	ELSIF byASCII=16#61 THEN	sOut_Single:='a';
	ELSIF byASCII=16#62 THEN  	sOut_Single:='b';
	ELSIF byASCII=16#63 THEN  	sOut_Single:='c';
	ELSIF byASCII=16#64 THEN	sOut_Single:='d';
	ELSIF byASCII=16#65 THEN	sOut_Single:='e';
	ELSIF byASCII=16#66 THEN	sOut_Single:='f';
	ELSIF byASCII=16#67 THEN	sOut_Single:='g';
	ELSIF byASCII=16#68 THEN	sOut_Single:='h';
	ELSIF byASCII=16#69 THEN	sOut_Single:='i';
	ELSIF byASCII=16#6A THEN	sOut_Single:='j';
	ELSIF byASCII=16#6B THEN	sOut_Single:='k';
	ELSIF byASCII=16#6C THEN	sOut_Single:='l';
	ELSIF byASCII=16#6D THEN	sOut_Single:='m';
	ELSIF byASCII=16#6E THEN	sOut_Single:='n';
	ELSIF byASCII=16#6F THEN	sOut_Single:='o';
	ELSIF byASCII=16#70 THEN	sOut_Single:='p';
	ELSIF byASCII=16#71 THEN	sOut_Single:='q';
	ELSIF byASCII=16#72 THEN	sOut_Single:='r';
	ELSIF byASCII=16#73 THEN	sOut_Single:='s';
	ELSIF byASCII=16#74 THEN	sOut_Single:='t';
	ELSIF byASCII=16#75 THEN	sOut_Single:='u';
	ELSIF byASCII=16#76 THEN	sOut_Single:='v';
	ELSIF byASCII=16#77 THEN	sOut_Single:='w';
	ELSIF byASCII=16#78 THEN	sOut_Single:='x';
	ELSIF byASCII=16#79 THEN	sOut_Single:='y';
	ELSIF byASCII=16#7A THEN	sOut_Single:='z';
	ELSIF byASCII=16#7B THEN	sOut_Single:='{';
	ELSIF byASCII=16#7C THEN	sOut_Single:='|';
	ELSIF byASCII=16#7D THEN	sOut_Single:='}';
	                                         
	ELSIF byASCII=16#30 THEN  	sOut_Single:='0';
	ELSIF byASCII=16#31 THEN  	sOut_Single:='1';
	ELSIF byASCII=16#32 THEN	sOut_Single:='2';
	ELSIF byASCII=16#33 THEN	sOut_Single:='3';
	ELSIF byASCII=16#34 THEN	sOut_Single:='4';
	ELSIF byASCII=16#35 THEN	sOut_Single:='5';
	ELSIF byASCII=16#36 THEN	sOut_Single:='6';
	ELSIF byASCII=16#37 THEN	sOut_Single:='7';
	ELSIF byASCII=16#38 THEN	sOut_Single:='8';
	ELSIF byASCII=16#39 THEN	sOut_Single:='9';
	ELSIF byASCII=16#3A THEN	sOut_Single:=':';
	ELSIF byASCII=16#3B THEN	sOut_Single:=';';
	ELSIF byASCII=16#3C THEN	sOut_Single:='<';
	ELSIF byASCII=16#3D THEN	sOut_Single:='=';
	ELSIF byASCII=16#3E THEN	sOut_Single:='>';
	ELSIF byASCII=16#3F THEN	sOut_Single:='?';
	ELSIF byASCII=16#40 THEN	sOut_Single:='@';
		                                     
	ELSIF byASCII=16#21 THEN	sOut_Single:='!';
	ELSIF byASCII=16#22 THEN	sOut_Single:='"';
	ELSIF byASCII=16#23 THEN	sOut_Single:='#';
//	ELSIF byASCII=16#24 THEN	sOut_Single:='$';
	ELSIF byASCII=16#25 THEN	sOut_Single:='%';
	ELSIF byASCII=16#26 THEN	sOut_Single:='&';
//	ELSIF byASCII=16#27 THEN	sOut_Single:=''';
	ELSIF byASCII=16#28 THEN	sOut_Single:='(';
	ELSIF byASCII=16#29 THEN	sOut_Single:=')';
	ELSIF byASCII=16#2A THEN	sOut_Single:='*';
	ELSIF byASCII=16#2B THEN	sOut_Single:='+';
	ELSIF byASCII=16#2C THEN	sOut_Single:=',';
	ELSIF byASCII=16#2D THEN	sOut_Single:='-';
	ELSIF byASCII=16#2E THEN	sOut_Single:='.';
	ELSIF byASCII=16#2F THEN	sOut_Single:='/';
	ELSE
		;	 //错误标志
	END_IF

END_FUNCTION_BLOCK

// Device/Application/PLC_PRG
PROGRAM PLC_PRG
VAR
	//(bHomingDone AND XRAY_RS485.Main_Step=20) OR Entity_IO.bEmergencyStop
	count: BYTE;
	bOver: BOOL; //关机结束指令
	bDebug_Laser:BOOL;
	TOF_Laser	:TOF;//激光灯控制
	TP_Laser	:TP;
	F_TRIG1		:F_TRIG;//激光灯按钮关闭
	R_TRIG1		:R_TRIG;//激光灯按钮关闭
	TOF_ET:TIME;
	TOF_PowerDelay: TOF;//延迟断电继电器控制
	LS_GetIPAddress_1: LS_GetIPAddress;
	LS_SetIPAddress_1: LS_SetIPAddress;
	rPLC_Load:REAL;
	LS_SetDintDT_1:LS_SysLib.LS_SetDintDT;
	bSetSysTime:BOOL;
	LS_ReadDintDT_1:LS_SysLib.LS_ReadDintDT;
	
	TON_StopScan:TON;

	iValidTrigger:UINT;
	iHopeNumPulse:UINT:=108;
	
	Step_Idle:INT;//待机模式下工作步骤
	Step_Scout:INT;//定位片模式下工作步骤
	Step_CBCT:INT;//CBCT模式下工作步骤
	Step_QuickScan:INT;//快速扫描下的工作步骤
	Step_DR:INT;//DR的工作步骤
	Step_XZ:INT;//XZ的工作步骤
	Step_AutoDR:INT;//自动空气校正DR
	bPulseOneStop	:BOOL;
	bScoutLast,bCBCTLast:BOOL;//最后一次扫描标志位

	TON_S30,TON_S40,TON_S41,TON_S42,TON_S43,TON_S50,TON_S52,TON_S60,TON_S70,TON_S80,TON_S90,TON_S44:TON;
	TON_S20_ABS,TON_S70_ABSX,TON_S70_ABSQ:TON;
	TOF_S40,TOF_S50:Standard.TOF;
	bXaryTwo_TEMP:BOOL; //二档输出中间变量
	
	TON_I00,TON_I10,TON_I20,TON_I30,TON_I40,TON_I50:Standard.TON;
	TON_C10,TON_C20,TON_C30,TON_C40,TON_C50,TON_C60,TON_C70,TON_C72,TON_C79,TON_C80,TON_C90,TON_C100,TON_C80_ABS,TON_C20_ABS:TON;
	TON_C210,TON_C201,TON_C220,TON_C230,TON_C240,TON_C250:TON;
	TOF_C80:Standard.TOF;
	R_TRIG_C20,R_TRIG_C220,R_TRIG_Jog,R_MoveRecordPos,R_RelStop:Standard.R_TRIG;
	F_TRIG_C20,F_TRIG_Jog:Standard.F_TRIG;
	
	AAA:STRING:='QWE';
	bSelfOK: BOOL;
	HandSelfStep: INT;
	bErrorReset:BOOL;
	TON_Error:TON;
	bHomingDone: BOOL;
	
	bGetPLC_IP,bSetPLC_IP,bGetPLC_Load:BOOL;
	
	TON_Home,TON_Home1:TON;
	
	bTestXayOne: BOOL;
	bTestXayTwo: BOOL;

	C_100: BOOL;
	bTCP_Socket:BOOL;
	TOF_JOG:TOF;
	bTestTrigger: BOOL;
	
	XZ_Velocity:REAL:=10;//设置不扫描时快速到扫描位的速度
	bTestTrigger11: BOOL;
	bTestTrigger22: BOOL;
	
	CTBOX_TON1:Standard.TON;
	CTBOX_TOF1:Standard.TOF;
	
	TON_IDLE:TON;
	bCBCT_AUTO_Manual:BOOL;//自动扫，手动扫标志位
	
	
	EncoderNum1,iStartTrigger1:UDINT;
	DB_EncoderNum1:UDINT;		//差值
	R_TRIG_debug,R_TRIG_debug2:R_TRIG;
	iActNumPulse1:UINT;//有效触发次数
	
	iSamplingRate1: INT:=2400;
	
	iHopePulse1:UINT;
	deubg_out:BOOL;
END_VAR

VAR PERSISTENT RETAIN
	rBedRecordHeight:REAL;//断电保存
	rBedRecordLength:REAL;//断电保存
END_VAR

VAR_OUTPUT	
	LampCmd5,LampCmd6,LampCmd7,LampCmd8:E_LampCmd;
END_VAR

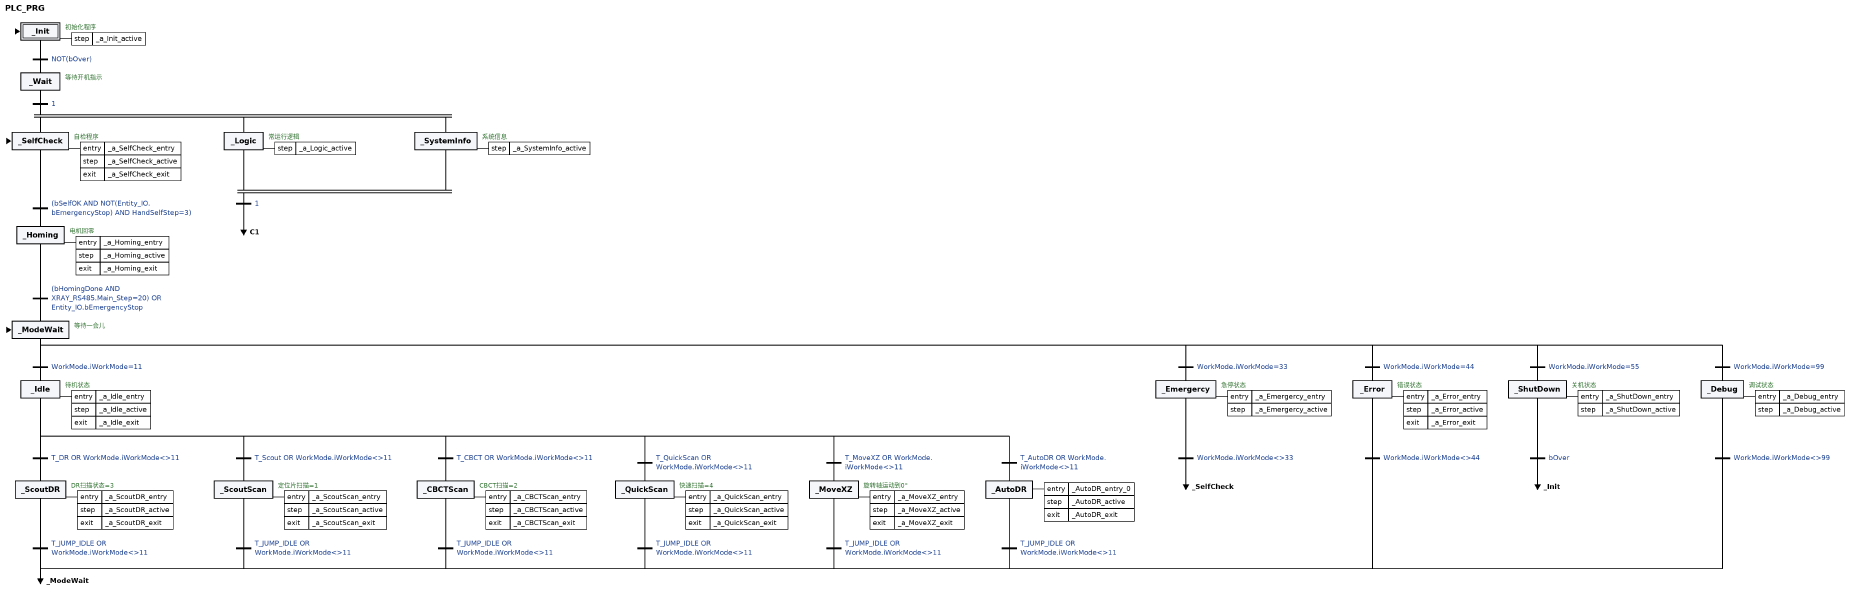
// 初始化程序
INITIAL_STEP _Init:
    _a_Init_active(N);  // step action
END_STEP
TRANSITION FROM _Init TO _Wait
    := NOT(bOver);
END_TRANSITION
// 等待开机指示
STEP _Wait:
END_STEP
TRANSITION FROM _Wait TO (_SelfCheck, _Logic, _SystemInfo)
    := 1;
END_TRANSITION
// 自检程序
STEP _SelfCheck:
    _a_SelfCheck_entry(P1);  // entry action
    _a_SelfCheck_active(N);  // step action
    _a_SelfCheck_exit(P0);  // exit action
END_STEP
TRANSITION FROM _SelfCheck TO _Homing
    := (bSelfOK AND NOT(Entity_IO.bEmergencyStop) AND HandSelfStep=3);
END_TRANSITION
// 电机回零
STEP _Homing:
    _a_Homing_entry(P1);  // entry action
    _a_Homing_active(N);  // step action
    _a_Homing_exit(P0);  // exit action
END_STEP
TRANSITION FROM _Homing TO _ModeWait
    := (bHomingDone AND XRAY_RS485.Main_Step=20) OR Entity_IO.bEmergencyStop;
END_TRANSITION
// 等待一会儿
STEP _ModeWait:
END_STEP
TRANSITION FROM _ModeWait TO _Idle
    := WorkMode.iWorkMode=11;
END_TRANSITION
// 待机状态
STEP _Idle:
    _a_Idle_entry(P1);  // entry action
    _a_Idle_active(N);  // step action
    _a_Idle_exit(P0);  // exit action
END_STEP
TRANSITION FROM _Idle TO _ScoutDR
    := T_DR OR WorkMode.iWorkMode<>11;
END_TRANSITION
// DR扫描状态=3
STEP _ScoutDR:
    _a_ScoutDR_entry(P1);  // entry action
    _a_ScoutDR_active(N);  // step action
    _a_ScoutDR_exit(P0);  // exit action
END_STEP
TRANSITION FROM _ScoutDR TO _ModeWait
    := T_JUMP_IDLE OR WorkMode.iWorkMode<>11;
END_TRANSITION
TRANSITION FROM _Idle TO _ScoutScan
    := T_Scout OR WorkMode.iWorkMode<>11;
END_TRANSITION
// 定位片扫描=1
STEP _ScoutScan:
    _a_ScoutScan_entry(P1);  // entry action
    _a_ScoutScan_active(N);  // step action
    _a_ScoutScan_exit(P0);  // exit action
END_STEP
TRANSITION FROM _ScoutScan TO _ModeWait
    := T_JUMP_IDLE OR WorkMode.iWorkMode<>11;
END_TRANSITION
TRANSITION FROM _Idle TO _CBCTScan
    := T_CBCT OR WorkMode.iWorkMode<>11;
END_TRANSITION
// CBCT扫描=2
STEP _CBCTScan:
    _a_CBCTScan_entry(P1);  // entry action
    _a_CBCTScan_active(N);  // step action
    _a_CBCTScan_exit(P0);  // exit action
END_STEP
TRANSITION FROM _CBCTScan TO _ModeWait
    := T_JUMP_IDLE OR WorkMode.iWorkMode<>11;
END_TRANSITION
TRANSITION FROM _Idle TO _QuickScan
    := T_QuickScan OR WorkMode.iWorkMode<>11;
END_TRANSITION
// 快速扫描=4
STEP _QuickScan:
    _a_QuickScan_entry(P1);  // entry action
    _a_QuickScan_active(N);  // step action
    _a_QuickScan_exit(P0);  // exit action
END_STEP
TRANSITION FROM _QuickScan TO _ModeWait
    := T_JUMP_IDLE OR WorkMode.iWorkMode<>11;
END_TRANSITION
TRANSITION FROM _Idle TO _MoveXZ
    := T_MoveXZ OR WorkMode.iWorkMode<>11;
END_TRANSITION
// 旋转轴运动到0°
STEP _MoveXZ:
    _a_MoveXZ_entry(P1);  // entry action
    _a_MoveXZ_active(N);  // step action
    _a_MoveXZ_exit(P0);  // exit action
END_STEP
TRANSITION FROM _MoveXZ TO _ModeWait
    := T_JUMP_IDLE OR WorkMode.iWorkMode<>11;
END_TRANSITION
TRANSITION FROM _Idle TO _AutoDR
    := T_AutoDR OR WorkMode.iWorkMode<>11;
END_TRANSITION
STEP _AutoDR:
    _AutoDR_entry_0(P1);  // entry action
    _AutoDR_active(N);  // step action
    _AutoDR_exit(P0);  // exit action
END_STEP
TRANSITION FROM _AutoDR TO _ModeWait
    := T_JUMP_IDLE OR WorkMode.iWorkMode<>11;
END_TRANSITION
TRANSITION FROM _ModeWait TO _Emergercy
    := WorkMode.iWorkMode=33;
END_TRANSITION
// 急停状态
STEP _Emergercy:
    _a_Emergercy_entry(P1);  // entry action
    _a_Emergercy_active(N);  // step action
END_STEP
TRANSITION FROM _Emergercy TO _SelfCheck
    := WorkMode.iWorkMode<>33;
END_TRANSITION
TRANSITION FROM _ModeWait TO _Error
    := WorkMode.iWorkMode=44;
END_TRANSITION
// 错误状态
STEP _Error:
    _a_Error_entry(P1);  // entry action
    _a_Error_active(N);  // step action
    _a_Error_exit(P0);  // exit action
END_STEP
TRANSITION FROM _Error TO _ModeWait
    := WorkMode.iWorkMode<>44;
END_TRANSITION
TRANSITION FROM _ModeWait TO _ShutDown
    := WorkMode.iWorkMode=55;
END_TRANSITION
// 关机状态
STEP _ShutDown:
    _a_ShutDown_entry(P1);  // entry action
    _a_ShutDown_active(N);  // step action
END_STEP
TRANSITION FROM _ShutDown TO _Init
    := bOver;
END_TRANSITION
TRANSITION FROM _ModeWait TO _Debug
    := WorkMode.iWorkMode=99;
END_TRANSITION
// 调试状态
STEP _Debug:
    _a_Debug_entry(P1);  // entry action
    _a_Debug_active(N);  // step action
END_STEP
TRANSITION FROM _Debug TO _ModeWait
    := WorkMode.iWorkMode<>99;
END_TRANSITION
// 常运行逻辑
STEP _Logic:
    _a_Logic_active(N);  // step action
END_STEP
// 系统信息
STEP _SystemInfo:
    _a_SystemInfo_active(N);  // step action
END_STEP
TRANSITION FROM (_Logic, _SystemInfo) TO (_Logic, _SystemInfo)
    := 1;
END_TRANSITION
// branch label C1
// branch label B1

ACTION _a_SelfCheck_active:

GVL_State.iPLC_State:=20;

(*目前只检查电机错误*)
	bSelfOK:=NOT(Axis_QJ.QJ_AxisState.bAxisErr OR Axis_XZ.XZ_AxisState.bAxisErr);

(*有错误自动复位*)	
	IF Entity_IO.bEmergencyStop = FALSE  THEN  //急停未被拍下
		CASE HandSelfStep OF
			0:
				IF Axis_QJ.QJ_AxisState.bAxisErr THEN
					Axis_QJ.QJ_AxisCmd.bReset:=TRUE;
				ELSE
					HandSelfStep:=1;
				END_IF
				
			1:
				IF Axis_XZ.XZ_AxisState.bAxisErr THEN
					Axis_XZ.XZ_AxisCmd.bReset:=TRUE;
				ELSE
					HandSelfStep:=2;
				END_IF
				
			2:
				Axis_XZ.XZ_AxisCmd.bReset:=FALSE;
				Axis_QJ.QJ_AxisCmd.bReset:=FALSE;
				HandSelfStep:=3;
				
			3:
				;	
		END_CASE
	END_IF;
	
(*旋转电机写入电机回零默认参数*)
	Axis_XZ.XZ_AxisCmd.AxisPara.rHomeAcc:=5.0;
	Axis_XZ.XZ_AxisCmd.AxisPara.iHomeMode:=10;
	Axis_XZ.XZ_AxisCmd.AxisPara.rHomeHighSpeed:=10;
	Axis_XZ.XZ_AxisCmd.AxisPara.rHomeLowSpeed:=5;
	
(*前进写入电机回零默认参数*)
	Axis_QJ.QJ_AxisCmd.AxisPara.rHomeAcc:=5.0;
	Axis_QJ.QJ_AxisCmd.AxisPara.iHomeMode:=10;
	Axis_QJ.QJ_AxisCmd.AxisPara.rHomeHighSpeed:=10;
	Axis_QJ.QJ_AxisCmd.AxisPara.rHomeLowSpeed:=5;
END_ACTION

ACTION _a_MoveXZ_entry:

GVL_State.iPLC_State:=52;//告诉上位机52，机架运动到位0位置
Step_XZ:=0; 
bTCP_Socket:=TRUE;
GVL_SCAN.bEnableScout:=FALSE;
GVL_SCAN.bEnableTrigger:=FALSE;
END_ACTION

ACTION _a_QuickScan_exit:


	LampCmd5:=E_LampCmd.关闭;
	LampCmd6:=E_LampCmd.关闭;
	LampCmd7:=E_LampCmd.关闭;
	LampCmd8:=E_LampCmd.关闭;
	
	Entity_IO.bTriggerPannel:=FALSE;
	Entity_IO.bTriggerOut:=FALSE;
	
	GVL_State.bEnable_CTBOX:=FALSE;//关闭CTBOX发送灯使能
END_ACTION

TRANSITION T_JUMP_IDLE:


	(*跳转到待机指令*)
	(*1.手动终止扫描，上位机发送终止扫描，扫描结束*)
	TON_StopScan.Q 
	OR (WorkStation_TCP.PLC_RECV1.m_nControlState>=1 AND WorkStation_TCP.PLC_RECV1.m_nSocketType=1)
	OR GVL_SCAN.bJumpScan;
END_TRANSITION

ACTION _a_ScoutDR_active:


	CASE Step_DR OF
		0:	//初始化准备流程
			(*1.给上位机发送的数据*)
			WorkStation_TCP.PLC_SEND1.m_nMoveState:=0;			//send[9]
			Axis_XZ.XZ_AxisCmd.bAbs:=FALSE;
			bTCP_Socket:=FALSE;
			bScoutLast := FALSE;
			
			(*2.运动准备数据*)
			(*2.1 写入旋转速度参数*)
			Axis_XZ.XZ_AxisCmd.AxisPara.rAbsVelocity:=36;//定位像扫描按照设定速度运动
			
			TON_S20_ABS(IN:=FALSE);
			Step_DR:=10;
		
		10:	//运动过程中变量复位标志
			TON_S30(IN:= FALSE );
			TON_S40(IN:= FALSE);TON_S50(IN:= FALSE);
			TON_S70(IN:= FALSE);TON_S80(IN:= FALSE);
			TOF_S50(IN:= FALSE);TON_S60(IN:= FALSE);
			TON_S52(IN:= FALSE );TON_S41(IN:=FALSE);
			TON_S43(IN:= FALSE );TON_S20_ABS(IN:=FALSE);	
			Axis_XZ.XZ_AxisCmd.bAbs:=FALSE;
			Step_DR:=20;
			
		20://开启运动
			(*1.给上位机发送的数据*)
			WorkStation_TCP.PLC_SEND1.m_nExpStates	:=1;//为曝光状态，枚举值，0:idle（空闲） 1:prep（训机） 2: ready（训机结束，准备完成，可以出束） 3: XrayOn（出射线） 4:XrayOff（关射线） 5 error；
			WorkStation_TCP.PLC_SEND1.m_nMoveState	:=0;//起始、终止状态， 默认值-1， 0为当前扫描方案（与常规意义不同，注意区别）处于准备好状态，可以准备扫描；1为当前扫描方案结束，运动过程中值为-1
			WorkStation_TCP.PLC_SEND1.m_nScanProType:=2;//执行扫描方案的类型，0为自动扫描，1为手动扫描，2为无设置意义的值，默认值为2
	
			(*2.旋转轴运动*)
			Axis_XZ.XZ_AxisCmd.AxisPara.rAbsPosition:=LIMIT(-4,WorkStation_TCP.PLC_RECV1.m_nRotateBegin,363);
			TON_S20_ABS(IN:= TRUE, PT:=T#1S );
			Axis_XZ.XZ_AxisCmd.bAbs:=TON_S20_ABS.Q;
			
			(*3.跳转下一个步骤*)	
			IF  ABS(Axis_XZ.XZ_AxisState.rActPosition-WorkStation_TCP.PLC_RECV1.m_nRotateBegin)<=1 THEN 
				Step_DR:=21;
			END_IF
				
		21://射线源参数写入成功标志
			TON_S20_ABS(IN:=FALSE);
			Axis_XZ.XZ_AxisCmd.bAbs:=FALSE;
			IF XRAY_RS485.Standby_Step=60 THEN		(*增加射线源参数写入成功标志*)
				Step_DR:=30;
			END_IF

		30: //开启7灯闪烁
			(*1.给上位机数据*)
			WorkStation_TCP.PLC_SEND1.m_nMoveState:=1;			//send[9]
			TON_S30(IN:=TRUE , PT:=T#1S , Q=> , ET=> );
			
			(*2.7灯闪烁*)
			GVL_State.bEnable_CTBOX:=TRUE;//开启CTBOX发送灯的状态
			LampCmd7:=E_LampCmd.慢闪;
			WorkStation_TCP.PLC_SEND1.m_nFocus:=7;//按键提示0228
			
			(*3.跳转*)
			IF TON_S30.Q THEN
				Step_DR:=31;
			END_IF
			
		31:
			GVL_State.bEnable_CTBOX:=FALSE;//关闭CTBOX发送灯的状态
			Step_DR:=40;
		
		40://等待用户按7键。此时7灯一直在闪烁
			(*1.发送上位机状态*)
			IF CTBOX_RS232.CTBOX_KEY_Manual THEN
				WorkStation_TCP.PLC_SEND1.m_nScanProType:=1;//执行扫描方案的类型，0为自动扫描，1为手动扫描，2为无设置意义的值，默认值为2
			END_IF
			
			(*2.7灯关闭*)
			TON_S41(IN:=(WorkStation_TCP.PLC_SEND1.m_nScanProType=1) , PT:=T#100MS , Q=> , ET=> );
			IF TON_S41.Q THEN
				LampCmd7:=E_LampCmd.关闭;  		//7灯关闭
				WorkStation_TCP.PLC_SEND1.m_nFocus:=0;//关闭按键提示0228
			END_IF
			
			TON_S42(IN:=FALSE , Q=> , ET=> );	//复位
			TON_S43(IN:=FALSE , Q=> , ET=> );	//复位
			
			(*3.跳转*)
			TON_S40(IN:= (WorkStation_TCP.PLC_SEND1.m_nScanProType=1), PT:=T#1S , Q=> , ET=> );
			IF TON_S40.Q THEN
				Step_DR:=41;
			END_IF
			
		41://中间状态清零，特别是从80跳转过来的变量清零
			GVL_State.bEnable_CTBOX:=FALSE;//关闭CTBOX发送灯的状态
			TON_S41(IN:=FALSE);TON_S80(IN:=FALSE);
			Entity_IO.bXaryOne:=FALSE;
			GVL_SCAN.bEnableTrigger:=FALSE;
			GVL_State.bScoutSecond:=TRUE;
			IF XRAY_RS485.Standby_Step=60 THEN
				Step_DR:=42;
			END_IF;	

		42:
			(*1.开启透视*)
			Entity_IO.bXaryOne:=TRUE;		//开启透视
			
			IF ABS(Axis_XZ.XZ_AxisState.rActPosition-WorkStation_TCP.PLC_RECV1.m_nAngleStart)<1 THEN
				GVL_SCAN.bEnableScout:=TRUE;	
			ELSE
				GVL_SCAN.bEnableScout:=FALSE;
			END_IF
			
			(*2.跳转指令*)
			TON_S43(IN:= Entity_IO.bXaryOne, PT:=T#1S , Q=> , ET=> );
			IF TON_S43.Q THEN
				IF XRAY_RS485.Rad_Step>=20 THEN  //此时射线源收到  =20
					Step_DR:=50;
				END_IF
			ELSE
			;
			END_IF;
			
			(*3.判断是否最后一次扫描标志位*)
			IF WorkStation_TCP.PLC_RECV1.m_nLastMsg=1 THEN
				bScoutLast := TRUE;
			ELSE
				bScoutLast := FALSE;
			END_IF 
			
			(*4.一二档信号超时报警，射线源30秒连续开启曝光会报警*)
			TON_S42(IN:=Entity_IO.bXaryOne , PT:=T#60S , Q=> , ET=> );
			IF TON_S42.Q THEN
				Step_DR:=44;	
			END_IF
			
		44:
			Entity_IO.bXaryOne:=FALSE;
			GVL_SCAN.bJumpScan:=TRUE;		//结束扫描，射线源超时报警了，EL019，结束扫描
			Step_DR:=44;	

		50://固定位置直接曝光28次
			TON_S43(IN:=FALSE , Q=> , ET=> );	//复位
			(*1.发送给上位机的数据*)
			WorkStation_TCP.PLC_SEND1.m_nMoveState	:=2;			//send[9]//0-准备过程中 1-准备完成 2-曝光中 3-本次扫描结束	
			WorkStation_TCP.PLC_SEND1.m_nScanProType:=2;			//send[16]
			
			(*2.开启允许曝光指令*)
			IF Entity_IO.bXaryOne AND ABS(Axis_XZ.XZ_AxisState.rActPosition-WorkStation_TCP.PLC_RECV1.m_nAngleStart)<1 THEN //新增射线源状态位置
				GVL_SCAN.bEnableTrigger:=TRUE;
			ELSE
				GVL_SCAN.bEnableTrigger:=FALSE;
			END_IF
			
			(*3.此过程给固定时间4秒,处理扫描*)
			TON_S50(IN:=TRUE , PT:=T#4S);
			IF TON_S50.Q THEN
				Step_DR:=52;	
			END_IF
		
		52://出射线状态结束，采集射线源状态机信息 //增加2档信号8秒计时器清零操作
			TON_S52(IN:=NOT(Trigger_HaoboPannel.bScoutPulse) , PT:= T#3S );
			Entity_IO.bXaryOne:=NOT(TON_S52.Q);
			IF TON_S52.Q THEN
				IF XRAY_RS485.Main_Step=20 THEN
					Step_DR:=60;
				END_IF
			END_IF
			
		60://判断是否最后一次扫描，如是，直接跳到待机模式，如果不是，接着定位扫描 ，第一次定位像和第二次定位像不一样，增加了床的运动
			TON_S80(IN:=FALSE);
			Entity_IO.bXaryOne:=FALSE;
			Axis_QJ.QJ_AxisCmd.bAbs:=FALSE;
			Axis_XZ.XZ_AxisCmd.bAbs:=FALSE;	
			TON_S70_ABSQ(IN:=FALSE);TON_S70_ABSX(IN:=FALSE);
			TON_S60(IN:=TRUE , PT:=T#1600MS , Q=> , ET=> );//留些时间给上位机发送本次扫描结束方案标志
			WorkStation_TCP.PLC_SEND1.m_nMoveState:=3;		//send[9] //0-准备过程中 1-准备完成 2-曝光中 3-本次扫描结束	
			IF TON_S60.Q THEN
				IF (WorkStation_TCP.PLC_RECV1.m_nCircleIndex+1)>=(WorkStation_TCP.PLC_RECV1.m_nCircleCount) AND bScoutLast THEN 	//用于区分自动扫是否最后一次，此时=1，=1都等于1
					GVL_SCAN.bJumpScan:=TRUE;
				END_IF;
			END_IF
			
			IF WorkStation_TCP.PLC_RECV1.m_nSocketType=1 THEN //增加第二次运动判断，m_nSocketType=1 
				Step_DR:=70;
			END_IF
			
		70://上位机选择移动床位置，机架根据命令运动到位
			Axis_QJ.QJ_AxisCmd.AxisPara.rAbsPosition:=LIMIT(0,WorkStation_TCP.PLC_RECV1.m_fScanTop,900);
			Axis_QJ.QJ_AxisCmd.AxisPara.rAbsVelocity:=50; //单位mm/s
			TON_S70_ABSQ(IN:=TRUE , PT:=T#1S , Q=> , ET=> );
			Axis_QJ.QJ_AxisCmd.bAbs:=TON_S70_ABSQ.Q;
			
			Axis_XZ.XZ_AxisCmd.AxisPara.rAbsPosition:=LIMIT(-4,WorkStation_TCP.PLC_RECV1.m_nRotateBegin,363);
			TON_S70_ABSX(IN:=TRUE , PT:=T#1S , Q=> , ET=> );
			Axis_XZ.XZ_AxisCmd.bAbs:=TON_S70_ABSX.Q;
			
			IF ABS(Axis_QJ.QJ_AxisState.rActPosition-WorkStation_TCP.PLC_RECV1.m_fScanTop)<1 AND ABS(Axis_XZ.XZ_AxisState.rActPosition-WorkStation_TCP.PLC_RECV1.m_nRotateBegin)<1 THEN
				WorkStation_TCP.PLC_SEND1.m_nMoveState:=1;		//send[9] //0-准备过程中 1-准备完成 2-曝光中 3-本次扫描结束	
			ELSE
				WorkStation_TCP.PLC_SEND1.m_nMoveState:=0;		//send[9] //0-准备过程中 1-准备完成 2-曝光中 3-本次扫描结束	
			END_IF
			
			TON_S70(IN:=ABS(Axis_QJ.QJ_AxisState.rActPosition-WorkStation_TCP.PLC_RECV1.m_fScanTop)<1 
					AND ABS(Axis_XZ.XZ_AxisState.rActPosition-WorkStation_TCP.PLC_RECV1.m_nRotateBegin)<1, 
					PT:=T#2S , Q=> , ET=> );//给你2秒走到位
			IF TON_S70.Q THEN
				Step_DR:=80;
			END_IF
		
		80://准备跳转，中间变量复位
			TOF_S50(IN:= FALSE);TON_S60(IN:= FALSE);TON_S70(IN:= FALSE);
			TON_S41(IN:= FALSE);TON_S42(IN:= FALSE);
			TON_S70_ABSQ(IN:=FALSE);TON_S70_ABSX(IN:=FALSE);
			Axis_QJ.QJ_AxisCmd.bAbs:=FALSE;
			Axis_XZ.XZ_AxisCmd.bAbs:=FALSE;
			TON_S80(IN:=TRUE , PT:= T#1S, Q=> , ET=> );
			IF TON_S80.Q THEN
				Step_DR:=41;
			END_IF;	
	END_CASE
END_ACTION

ACTION _a_Idle_exit:


	Step_Idle:=0;
	
	LampCmd5:=E_LampCmd.关闭;
	LampCmd6:=E_LampCmd.关闭;
	LampCmd7:=E_LampCmd.关闭;
	LampCmd8:=E_LampCmd.关闭;
	
	GVL_State.bBooting:=FALSE;
END_ACTION

TRANSITION T_DR:

(*进入dr扫描*)
	WorkStation_TCP.PLC_RECV1.m_nSocketType=1 AND WorkStation_TCP.PLC_RECV1.m_nExpId=3
END_TRANSITION

ACTION _AutoDR_exit:


	LampCmd5:=E_LampCmd.关闭;
	LampCmd6:=E_LampCmd.关闭;
	LampCmd7:=E_LampCmd.关闭;
	LampCmd8:=E_LampCmd.关闭;
	
	Entity_IO.bTriggerPannel:=FALSE;
	Entity_IO.bTriggerOut:=FALSE;
END_ACTION

ACTION _a_Idle_entry:


	Step_Idle:=0; //
	bPulseOneStop:=TRUE;
	
	GVL_SCAN.bJumpScan:=FALSE;
	
	Axis_XZ.XZ_AxisCmd.bAbs:=FALSE;
	Axis_QJ.QJ_AxisCmd.bAbs:=FALSE;
	
	Axis_QJ.QJ_AxisCmd.bStop:=FALSE;
	Axis_XZ.XZ_AxisCmd.bStop:=FALSE;
		
	Axis_XZ.XZ_AxisCmd.bReset:=FALSE;
	Axis_QJ.QJ_AxisCmd.bReset:=FALSE;
	
	GVL_SCAN.bEnableTrigger:=FALSE;
	GVL_State.bBooting:=TRUE;
	
	WorkStation_TCP.PLC_SEND1.m_nFocus:=0;//按键提示

	Step_CBCT:=0;
	Step_Scout:=0;
END_ACTION

ACTION _a_SelfCheck_exit:


Axis_QJ.QJ_AxisCmd.bSetHomePara:=TRUE;

Axis_XZ.XZ_AxisCmd.bSetHomePara:=TRUE;
END_ACTION

ACTION _a_Error_entry:

	bErrorReset:=TRUE;
	TON_Error(IN:=FALSE);
END_ACTION

TRANSITION T_QuickScan:


(*进入快速扫描*)
	WorkStation_TCP.PLC_RECV1.m_nSocketType=1 AND WorkStation_TCP.PLC_RECV1.m_nExpId=4 //这里需要上位机增加一个4,判断是快速扫描
END_TRANSITION

ACTION _AutoDR_active:

	CASE Step_AutoDR OF 
		0:	//初始化准备流程
			(*1.给上位机发送的数据*)
			WorkStation_TCP.PLC_SEND1.m_nMoveState:=0;			//send[9] //0-准备过程中 1-准备完成 2-曝光中 3-本次扫描结束
			bTCP_Socket:=FALSE; 
			bCBCTLast:=FALSE;
			
			(*2.运动准备数据*)
			(*2.1 写入旋转速度参数*)
		(*	IF WorkStation_TCP.PLC_RECV1.m_fSecondPerCicle<>0 THEN//避免除零
				Axis_XZ.XZ_AxisCmd.AxisPara.rAbsVelocity:=UDINT_TO_REAL(LIMIT(360/300 ,360/WorkStation_TCP.PLC_RECV1.m_fSecondPerCicle ,360/20 ));
				XZ_Velocity:=LIMIT(360/300 ,360/UDINT_TO_REAL(WorkStation_TCP.PLC_RECV1.m_fSecondPerCicle) ,360/20);
			ELSE
				Axis_XZ.XZ_AxisCmd.AxisPara.rAbsVelocity:=8;
			END_IF;
		*)
			Axis_XZ.XZ_AxisCmd.AxisPara.rAbsVelocity:=36;
			Step_AutoDR:=10;

		10:	//运动过程中变量复位标志
			TON_C20(IN:= FALSE);TON_C30(IN:= FALSE);
			TON_C40(IN:= FALSE);TON_C50(IN:= FALSE);TON_C60(IN:= FALSE);
			TON_C70(IN:= FALSE);TON_C80(IN:= FALSE);TON_C72(IN:=FALSE);
			TON_C210(IN:= FALSE);TON_C220(IN:= FALSE);TON_C230(IN:= FALSE);
			TON_C240(IN:= FALSE);TON_C250(IN:= FALSE);
			TON_C20_ABS(IN:=FALSE);
			TOF_C80(IN:= FALSE);
			Axis_XZ.XZ_AxisCmd.bAbs:=FALSE;
			Step_AutoDR:=20;
			
		20://按5键，移动床到预设位置，松开即停，机架直接到预设位置
			(*1.发送给上位机的数据*)
			WorkStation_TCP.PLC_SEND1.m_nExpStates:=1;		//0-准备过程中 1-准备完成 2-曝光中 3-本次扫描结束	
			WorkStation_TCP.PLC_SEND1.m_nMoveState:=0;		//起始、终止状态， 默认值0， 1为当前扫描方案处于准备好状态，可以准备扫描；2为当前扫描方案结束，运动过程中值为0
			WorkStation_TCP.PLC_SEND1.m_nScanProType:=2;	//扫描方案类型 , 1-手动，0-自动. 
			
			(*2.旋转轴直接运动到目标位置*)
			Axis_XZ.XZ_AxisCmd.AxisPara.rAbsPosition:=LIMIT(-3,WorkStation_TCP.PLC_RECV1.m_nRotateBegin,363);
			Axis_XZ.XZ_AxisCmd.AxisPara.rAbsVelocity:=36;
			TON_C20_ABS(IN:=TRUE , PT:=T#1S);
			Axis_XZ.XZ_AxisCmd.bAbs:=TON_C20_ABS.Q;
			
			(*3.前进轴运动*)
			R_TRIG_C20(CLK:= CTBOX_RS232.CTBOX_KEY_MoveDistance, Q=> );//触发运动
			F_TRIG_C20(CLK:= CTBOX_RS232.CTBOX_KEY_MoveDistance, Q=> );//触发停止
			
			Axis_QJ.QJ_AxisCmd.bAbs	:=R_TRIG_C20.Q;
			Axis_QJ.QJ_AxisCmd.AxisPara.rAbsPosition	:=LIMIT(0,WorkStation_TCP.PLC_RECV1.m_fScanTop,900);
			Axis_QJ.QJ_AxisCmd.bStop:=F_TRIG_C20.Q;
			
			(*4.5灯逻辑处理*)
			GVL_State.bEnable_CTBOX:=TRUE;//开启CTBOX发送灯使能
			IF ABS(Axis_QJ.QJ_AxisState.rActPosition-WorkStation_TCP.PLC_RECV1.m_fScanTop)>1 THEN
				LampCmd5:=E_LampCmd.慢闪;
				WorkStation_TCP.PLC_SEND1.m_nFocus:=5;//按键提示0228
			ELSE
				LampCmd5:=E_LampCmd.关闭;
				WorkStation_TCP.PLC_SEND1.m_nFocus:=0;//关闭按键提示0228
			END_IF
			
			(*5.跳转*)
			TON_C20(IN:=ABS(Axis_QJ.QJ_AxisState.rActPosition-WorkStation_TCP.PLC_RECV1.m_fScanTop)<1 
				AND ABS(Axis_XZ.XZ_AxisState.rActPosition-WorkStation_TCP.PLC_RECV1.m_nRotateBegin)<1 , PT:=T#2S);
			IF TON_C20.Q THEN  
				Step_AutoDR:=30;
			END_IF
			
		30:	//射线源参数写入成功标志
			TON_C20_ABS(IN:=FALSE);
			LampCmd5:=E_LampCmd.关闭;
			Axis_XZ.XZ_AxisCmd.bAbs:=FALSE;
			Axis_QJ.QJ_AxisCmd.bAbs:=FALSE;
			Axis_QJ.QJ_AxisCmd.bStop:=FALSE;
			IF XRAY_RS485.Standby_Step=60 THEN
				Step_AutoDR:=40;
			END_IF
			
		40:	//7灯和8灯开始慢闪
			WorkStation_TCP.PLC_SEND1.m_nMoveState:=1;		//起始、终止状态， 默认值0， 1为当前扫描方案处于准备好状态
			LampCmd7:=E_LampCmd.慢闪;
			LampCmd8:=E_LampCmd.慢闪;
			WorkStation_TCP.PLC_SEND1.m_nFocus:=8;//按键提示0228
			TON_C40(IN:=TRUE , PT:=T#600MS , Q=> , ET=> );
			IF TON_C40.Q THEN
				Step_AutoDR:=41;
			END_IF
		41:
			GVL_State.bEnable_CTBOX:=FALSE;//开启CTBOX发送灯使能
			Step_AutoDR:=50;
			
		50://用户选择自动扫描或手动扫描
			IF CTBOX_RS232.CTBOX_KEY_Auto=FALSE AND CTBOX_RS232.CTBOX_KEY_Manual THEN
				WorkStation_TCP.PLC_SEND1.m_nScanProType:=1;								//扫描方案类型 , 1-手动，0-自动. 
				bCBCT_AUTO_Manual:=TRUE;
			ELSIF CTBOX_RS232.CTBOX_KEY_Auto AND CTBOX_RS232.CTBOX_KEY_Manual=FALSE THEN
				WorkStation_TCP.PLC_SEND1.m_nScanProType:=0;								//扫描方案类型 , 1-手动，0-自动. 
				bCBCT_AUTO_Manual:=FALSE;
			ELSIF CTBOX_RS232.CTBOX_KEY_Auto=FALSE AND CTBOX_RS232.CTBOX_KEY_Manual=FALSE THEN
				;
			ELSIF CTBOX_RS232.CTBOX_KEY_Auto AND CTBOX_RS232.CTBOX_KEY_Manual THEN
				;
			END_IF
			
			IF (CTBOX_RS232.CTBOX_KEY_Auto AND CTBOX_RS232.CTBOX_KEY_Manual=FALSE) OR CTBOX_RS232.CTBOX_KEY_Manual AND CTBOX_RS232.CTBOX_KEY_Auto=FALSE THEN
				Step_AutoDR:=60;
			END_IF
			
		60://7和8灯关闭 
			GVL_State.bEnable_CTBOX:=TRUE;
			LampCmd7:=E_LampCmd.关闭;
			LampCmd8:=E_LampCmd.关闭;
			WorkStation_TCP.PLC_SEND1.m_nFocus:=0;	//关闭按键提示0228
			TON_C60(IN:= TRUE, PT:=T#1S , Q=> , ET=> );
			
			IF TON_C60.Q THEN
				Step_AutoDR:=70;
			END_IF
			
		70://扫描中间态，给跳转用的
			GVL_State.bEnable_CTBOX:=FALSE;//关闭CTBOX发送灯使能
			WorkStation_TCP.PLC_SEND1.m_nMoveState	:=1;	//send[9]
			WorkStation_TCP.PLC_SEND1.m_nScanProType:=2;	//send[16]
			TON_C70(IN:=TRUE , PT:=T#2S , Q=> , ET=> );
			TON_C220(IN:=FALSE);TON_C72(IN:=FALSE);TON_S50(IN:=FALSE , PT:=T#4S);
			Axis_QJ.QJ_AxisCmd.bAbs:=FALSE;//复位前进轴
			Axis_XZ.XZ_AxisCmd.bAbs:=FALSE;//复位旋转轴
			TON_C72(IN:=FALSE);
			TON_C79(IN:=TRUE , PT:= T#1S, Q=> , ET=> );
			
			IF XRAY_RS485.Standby_Step=60 THEN  //保证写入参数
				Entity_IO.bXaryOne:=TRUE;//开启透视
			END_IF;
			
			(*判断是否最后一次扫描*)
			IF WorkStation_TCP.PLC_RECV1.m_nLastMsg=1 THEN
				bCBCTLast := TRUE;
			ELSE
				bCBCTLast := FALSE;
			END_IF
			
			(*跳转指令*)
			IF TON_C70.Q AND Entity_IO.bXaryOne THEN
				Step_AutoDR:=79;
			END_IF
			
		74:
			Entity_IO.bXaryOne:=FALSE;
			GVL_SCAN.bJumpScan:=TRUE;		//结束扫描，射线源超时报警了，EL019，结束扫描
			Step_AutoDR:=74;
			
		79:
			Axis_XZ.XZ_AxisCmd.bAbs:=FALSE;
			TON_C80_ABS(IN:=FALSE);
			TON_S50(IN:=FALSE , PT:=T#4S);
			TON_C79(IN:=TRUE , PT:= T#4S, Q=> , ET=> );
			IF TON_C79.Q THEN
				Step_AutoDR:=80;
			END_IF
			
			IF ABS(Axis_XZ.XZ_AxisState.rActPosition-WorkStation_TCP.PLC_RECV1.m_nAngleStart)<1 THEN
				GVL_SCAN.bEnableScout:=TRUE;	
			ELSE
				GVL_SCAN.bEnableScout:=FALSE;
			END_IF
			
		80://第一次自动扫描
			(*1.给上位机发送的数*)
			TON_C79(IN:=FALSE);
			WorkStation_TCP.PLC_SEND1.m_nMoveState	:=2;
			WorkStation_TCP.PLC_SEND1.m_nScanProType:=2;

			(*2.开启允许曝光指令*)
			IF Entity_IO.bXaryOne AND ABS(Axis_XZ.XZ_AxisState.rActPosition-WorkStation_TCP.PLC_RECV1.m_nAngleStart)<1 THEN //新增射线源状态位置
				GVL_SCAN.bEnableTrigger:=TRUE;
			ELSE
				GVL_SCAN.bEnableTrigger:=FALSE;
			END_IF
			
			(*3.此过程给固定时间4秒,处理扫描*)
			TON_S50(IN:=TRUE , PT:=T#4S);
			IF TON_S50.Q THEN
				Step_AutoDR:=81;	
			END_IF
			
			(*6.透视信号超时报警，射线源30秒连续开启曝光会报警*)
			TON_C72(IN:=Entity_IO.bXaryOne , PT:=T#1M , Q=> , ET=> );
			IF TON_C72.Q THEN
				Step_AutoDR:=74;	
			END_IF
			
		81://出射线状态结束，采集射线源状态机信息
			Entity_IO.bXaryOne		:=FALSE;
			TON_C90(IN:=FALSE , PT:=T#2S , Q=> , ET=> );
			IF XRAY_RS485.Main_Step=20 THEN
				Step_AutoDR:=90;
			END_IF
			
		90://中间变量清零1070
			Axis_XZ.XZ_AxisCmd.bAbs	:=FALSE;	
			Entity_IO.bXaryOne		:=FALSE;
			TON_C100(IN:= FALSE, PT:=T#2S);
			C_100:=FALSE;
			WorkStation_TCP.PLC_SEND1.m_nMoveState:=3; //send [9]
			TON_C90(IN:=TRUE , PT:=T#2S , Q=> , ET=> );
			IF TON_C90.Q THEN
				IF (WorkStation_TCP.PLC_RECV1.m_nCircleIndex+1)>=(WorkStation_TCP.PLC_RECV1.m_nCircleCount) AND bCBCTLast THEN //最后一次扫描退出
					GVL_SCAN.bJumpScan:=TRUE;
				END_IF
			END_IF
			
			C_100:=FALSE;
			TON_C80_ABS(IN:=FALSE);
			
			(*增加跳转判断*)
			IF WorkStation_TCP.PLC_RECV1.m_nSocketType=1 THEN 	//增加第二次运动判断，m_nSocketType=1 
				Step_AutoDR:=100;
			END_IF
			
		100:	
			C_100:=TRUE;
			(*延迟2秒*)
			TON_C100(IN:= C_100, PT:=T#1S);
			(*跳转*)
			IF TON_C100.Q THEN
				Step_AutoDR:=110;
			END_IF;
			
		110://CBCT下的自动扫还是手动扫，根据上位机命令
			TON_C210(IN:= FALSE);TON_C201(IN:=FALSE);
			C_100:=FALSE;
			
			IF WorkStation_TCP.PLC_RECV1.m_nScanUseType=1 THEN
				Step_AutoDR:=200;		//手动扫描
			ELSE
				Step_AutoDR:=120;		//自动扫描
			END_IF
		 
		120://开启自动扫描
			TOF_C80(IN:= FALSE);TON_C100(IN:=FALSE);TON_C90(IN:=FALSE);TON_C80(IN:=FALSE);TON_C70(IN:=FALSE);TON_C60(IN:=FALSE);
			Axis_QJ.QJ_AxisCmd.AxisPara.rAbsPosition:=LIMIT(0,WorkStation_TCP.PLC_RECV1.m_fScanTop,900);
			Axis_QJ.QJ_AxisCmd.bAbs:=TRUE;
			
			IF ABS(Axis_QJ.QJ_AxisState.rActPosition-Axis_QJ.QJ_AxisCmd.AxisPara.rAbsPosition)<1 THEN
				WorkStation_TCP.PLC_SEND1.m_nMoveState:=1; 			//send [9]
				Step_AutoDR:=70;				//自动扫描
			ELSE
				WorkStation_TCP.PLC_SEND1.m_nMoveState:=0; 			//send [9]	//0-准备过程中 1-准备完成 2-曝光中 3-本次扫描结束
			END_IF
			
		(*-------------------------手动扫描-----------------------------*)	
		200://中间状态清零
			WorkStation_TCP.PLC_SEND1.m_nMoveState:=0; //send [9]	//0-准备过程中 1-准备完成 2-曝光中 3-本次扫描结束
			Axis_XZ.XZ_AxisCmd.bAbs:=FALSE;
			Step_AutoDR:=201;

		201:
			TON_C201(IN:= TRUE, PT:=T#1S , Q=> , ET=> );
			IF TON_C201.Q THEN
				Step_AutoDR:=210;
			END_IF
			
		210://7灯闪烁，机架运动到目标位置
			(*1.发送给上位机的数据*)
			WorkStation_TCP.PLC_SEND1.m_nMoveState:=0; //send [9]	//0-准备过程中 1-准备完成 2-曝光中 3-本次扫描结束
			TON_C201(IN:= FALSE);
			(*2.7灯闪烁*)
			GVL_State.bEnable_CTBOX:=TRUE;			//开启CTBOX发送灯使能
			LampCmd7:=E_LampCmd.慢闪;
			WorkStation_TCP.PLC_SEND1.m_nFocus:=7;	//按键提示0228
			
			(*3.旋转轴运动到目标位置*)
			Axis_XZ.XZ_AxisCmd.AxisPara.rAbsPosition:=LIMIT(-4,WorkStation_TCP.PLC_RECV1.m_nRotateBegin,363);
			Axis_XZ.XZ_AxisCmd.AxisPara.rAbsVelocity:=XZ_Velocity;
			
			IF WorkStation_TCP.PLC_RECV1.m_nSocketType=1 THEN
				Axis_XZ.XZ_AxisCmd.bAbs:=TRUE;
			END_IF;
			
			(*4.到位后1秒跳转*)
			TON_C210(IN:=ABS(Axis_XZ.XZ_AxisState.rActPosition-WorkStation_TCP.PLC_RECV1.m_nRotateBegin)<1 , PT:=T#1S , Q=> , ET=> );
			IF TON_C210.Q THEN
				Step_AutoDR:=221;	
			END_IF
		
		221://中间状态清零
			Axis_XZ.XZ_AxisCmd.bAbs:=FALSE;
			Axis_QJ.QJ_AxisCmd.bAbs:=FALSE;
			GVL_State.bEnable_CTBOX:=FALSE;//关闭CTBOX发送灯使能
			Step_AutoDR:=220;
			
		220://用户按7键，床自动走到预设位置
			(*1.按7键关闭7灯*)
			IF CTBOX_RS232.CTBOX_KEY_Manual THEN
				LampCmd7:=E_LampCmd.关闭;
				GVL_State.bEnable_CTBOX:=TRUE;//开启CTBOX发送灯使能
				WorkStation_TCP.PLC_SEND1.m_nFocus:=0;	//关闭按键提示0228
			END_IF
			
			(*2.触发床运动*)
			R_TRIG_C220(CLK:=CTBOX_RS232.CTBOX_KEY_Manual , Q=> );
			Axis_QJ.QJ_AxisCmd.AxisPara.rAbsPosition:=LIMIT(0,WorkStation_TCP.PLC_RECV1.m_fScanTop,900);
			Axis_QJ.QJ_AxisCmd.bAbs:=R_TRIG_C220.Q;
			
			(*3.跳转指令*)
			IF ABS(Axis_QJ.QJ_AxisState.rActPosition-WorkStation_TCP.PLC_RECV1.m_fScanTop)<1 AND (LampCmd7=E_LampCmd.关闭) THEN //保证必须按下7键
				WorkStation_TCP.PLC_SEND1.m_nMoveState:=1; //send [9]	//0-准备过程中 1-准备完成 2-曝光中 3-本次扫描结束
			ELSE
				WorkStation_TCP.PLC_SEND1.m_nMoveState:=0; //send [9]	//0-准备过程中 1-准备完成 2-曝光中 3-本次扫描结束
			END_IF
			
			(*4.延迟跳转，保证send [9]发送*)
			TOF_C80(IN:= FALSE);TON_C100(IN:=FALSE);TON_C90(IN:=FALSE);TON_C80(IN:=FALSE);TON_C70(IN:=FALSE);TON_C60(IN:=FALSE);
			TON_C210(IN:=FALSE);TON_C72(IN:=FALSE);TON_C201(IN:=FALSE);
			TON_C220(IN:=(WorkStation_TCP.PLC_SEND1.m_nMoveState=1) , PT:=T#2S , Q=> , ET=> );
			IF TON_C220.Q THEN
				Step_AutoDR:=70;
			END_IF		
	END_CASE
END_ACTION

ACTION _a_QuickScan_entry:



GVL_State.iPLC_State:=65;//告诉上位机65，是快速扫描状态
Step_CBCT:=0; 
GVL_SCAN.bJumpScan:=FALSE;
bTCP_Socket:=TRUE;

GVL_SCAN.bEnableScout:=FALSE;
GVL_SCAN.bEnableTrigger:=FALSE;

GVL_State.bEnable_CTBOX:=FALSE;//进入使能CTBOX——Enable
END_ACTION

ACTION _a_Error_active:

	(*电机进行复位操作*)	
	IF bErrorReset THEN	
		IF Axis_XZ.XZ_AxisState.bAxisErr THEN
			Axis_XZ.XZ_AxisCmd.bReset:=TRUE;
		ELSE
			;		
		END_IF
		
		IF Axis_QJ.QJ_AxisState.bAxisErr THEN
			Axis_QJ.QJ_AxisCmd.bReset:=TRUE;
		ELSE
			;		
		END_IF
		bErrorReset:=FALSE;
	ELSE
		Axis_QJ.QJ_AxisCmd.bReset:=FALSE;
		Axis_XZ.XZ_AxisCmd.bReset:=FALSE;
	END_IF
	
	(*延迟2秒输出*)
	TON_Error(IN:=TRUE , PT:=T#2S , Q=> , ET=> );
	IF TON_Error.Q THEN
		GVL_State.iPLC_State:=80;
	END_IF
END_ACTION

TRANSITION T_AutoDR:


(*进入自动空气校正DR扫描*)
	WorkStation_TCP.PLC_RECV1.m_nSocketType=1 AND WorkStation_TCP.PLC_RECV1.m_nExpId=6
END_TRANSITION

ACTION _a_CBCTScan_exit:

	LampCmd5:=E_LampCmd.关闭;
	LampCmd6:=E_LampCmd.关闭;
	LampCmd7:=E_LampCmd.关闭;
	LampCmd8:=E_LampCmd.关闭;
	
	Entity_IO.bTriggerPannel:=FALSE;
	Entity_IO.bTriggerOut:=FALSE;
	
	GVL_State.bEnable_CTBOX:=FALSE;//关闭CTBOX发送灯使能
END_ACTION

ACTION _a_CBCTScan_active:

	CASE Step_CBCT OF 
		0:	//初始化准备流程
			(*1.给上位机发送的数据*)
			WorkStation_TCP.PLC_SEND1.m_nMoveState:=0;			//send[9] //0-准备过程中 1-准备完成 2-曝光中 3-本次扫描结束
			bTCP_Socket:=FALSE; 
			bCBCTLast:=FALSE;
			
			(*2.运动准备数据*)
			(*2.1 写入旋转速度参数*)
			IF WorkStation_TCP.PLC_RECV1.m_fSecondPerCicle<>0 THEN//避免除零
				Axis_XZ.XZ_AxisCmd.AxisPara.rAbsVelocity:=UDINT_TO_REAL(LIMIT(360/300 ,360/WorkStation_TCP.PLC_RECV1.m_fSecondPerCicle ,360/20 ));
				XZ_Velocity:=LIMIT(360/300 ,360/UDINT_TO_REAL(WorkStation_TCP.PLC_RECV1.m_fSecondPerCicle) ,360/20);
			ELSE
				Axis_XZ.XZ_AxisCmd.AxisPara.rAbsVelocity:=8;
			END_IF;
			GVL_State.bEnable_CTBOX:=FALSE;//关闭CTBOX发送灯使能
			Step_CBCT:=10;

		10:	//运动过程中变量复位标志
			TON_C20(IN:= FALSE);TON_C30(IN:= FALSE);
			TON_C40(IN:= FALSE);TON_C50(IN:= FALSE);TON_C60(IN:= FALSE);
			TON_C70(IN:= FALSE);TON_C80(IN:= FALSE);TON_C72(IN:=FALSE);
			TON_C210(IN:= FALSE);TON_C220(IN:= FALSE);TON_C230(IN:= FALSE);
			TON_C240(IN:= FALSE);TON_C250(IN:= FALSE);
			TON_C20_ABS(IN:=FALSE);
			TOF_C80(IN:= FALSE);
			Axis_XZ.XZ_AxisCmd.bAbs:=FALSE;
			Step_CBCT:=20;
			
		20://按5键，移动床到预设位置，松开即停，机架直接到预设位置
			(*1.发送给上位机的数据*)
			WorkStation_TCP.PLC_SEND1.m_nExpStates:=1;		//0-准备过程中 1-准备完成 2-曝光中 3-本次扫描结束	
			WorkStation_TCP.PLC_SEND1.m_nMoveState:=0;		//起始、终止状态， 默认值0， 1为当前扫描方案处于准备好状态，可以准备扫描；2为当前扫描方案结束，运动过程中值为0
			WorkStation_TCP.PLC_SEND1.m_nScanProType:=2;	//扫描方案类型 , 1-手动，0-自动. 
			
			(*2.旋转轴直接运动到目标位置*)
			Axis_XZ.XZ_AxisCmd.AxisPara.rAbsPosition:=LIMIT(-3,WorkStation_TCP.PLC_RECV1.m_nRotateBegin,363);
			Axis_XZ.XZ_AxisCmd.AxisPara.rAbsVelocity:=18;
			TON_C20_ABS(IN:=TRUE , PT:=T#1S);
			Axis_XZ.XZ_AxisCmd.bAbs:=TON_C20_ABS.Q;
			
			(*3.前进轴运动*)
			R_TRIG_C20(CLK:= CTBOX_RS232.CTBOX_KEY_MoveDistance, Q=> );//触发运动
			F_TRIG_C20(CLK:= CTBOX_RS232.CTBOX_KEY_MoveDistance, Q=> );//触发停止
			
			Axis_QJ.QJ_AxisCmd.bAbs	:=R_TRIG_C20.Q;
			Axis_QJ.QJ_AxisCmd.AxisPara.rAbsPosition	:=LIMIT(0,WorkStation_TCP.PLC_RECV1.m_fScanTop,900);
			Axis_QJ.QJ_AxisCmd.bStop:=F_TRIG_C20.Q;
			
			(*4.5灯逻辑处理*)
			GVL_State.bEnable_CTBOX:=TRUE;//开启CTBOX发送灯使能
			IF ABS(Axis_QJ.QJ_AxisState.rActPosition-WorkStation_TCP.PLC_RECV1.m_fScanTop)>1 THEN
				LampCmd5:=E_LampCmd.慢闪;
				WorkStation_TCP.PLC_SEND1.m_nFocus:=5;//按键提示0228
			ELSE
				LampCmd5:=E_LampCmd.关闭;
				WorkStation_TCP.PLC_SEND1.m_nFocus:=0;//关闭按键提示0228
			END_IF
			
			(*5.跳转*)
			TON_C20(IN:=ABS(Axis_QJ.QJ_AxisState.rActPosition-WorkStation_TCP.PLC_RECV1.m_fScanTop)<1 
				AND ABS(Axis_XZ.XZ_AxisState.rActPosition-WorkStation_TCP.PLC_RECV1.m_nRotateBegin)<1 , PT:=T#2S);
			IF TON_C20.Q THEN  
				Step_CBCT:=30;
			END_IF
			
		30:	//射线源参数写入成功标志
			TON_C20_ABS(IN:=FALSE);
			LampCmd5:=E_LampCmd.关闭;
			Axis_XZ.XZ_AxisCmd.bAbs:=FALSE;
			Axis_QJ.QJ_AxisCmd.bAbs:=FALSE;
			Axis_QJ.QJ_AxisCmd.bStop:=FALSE;
			IF XRAY_RS485.Standby_Step=60 THEN
				Step_CBCT:=40;
			END_IF
			
		40:	//7灯和8灯开始慢闪
			WorkStation_TCP.PLC_SEND1.m_nMoveState:=1;		//起始、终止状态， 默认值0， 1为当前扫描方案处于准备好状态
			LampCmd7:=E_LampCmd.慢闪;
			LampCmd8:=E_LampCmd.慢闪;
			WorkStation_TCP.PLC_SEND1.m_nFocus:=8;//按键提示0228
			TON_C40(IN:=TRUE , PT:=T#600MS , Q=> , ET=> );
			IF TON_C40.Q THEN
				Step_CBCT:=41;
			END_IF
		41:
			GVL_State.bEnable_CTBOX:=FALSE;//开启CTBOX发送灯使能
			Step_CBCT:=50;
			
		50://用户选择自动扫描或手动扫描
			IF CTBOX_RS232.CTBOX_KEY_Auto=FALSE AND CTBOX_RS232.CTBOX_KEY_Manual THEN
				WorkStation_TCP.PLC_SEND1.m_nScanProType:=1;								//扫描方案类型 , 1-手动，0-自动. 
				bCBCT_AUTO_Manual:=TRUE;
			ELSIF CTBOX_RS232.CTBOX_KEY_Auto AND CTBOX_RS232.CTBOX_KEY_Manual=FALSE THEN
				WorkStation_TCP.PLC_SEND1.m_nScanProType:=0;								//扫描方案类型 , 1-手动，0-自动. 
				bCBCT_AUTO_Manual:=FALSE;
			ELSIF CTBOX_RS232.CTBOX_KEY_Auto=FALSE AND CTBOX_RS232.CTBOX_KEY_Manual=FALSE THEN
				;
			ELSIF CTBOX_RS232.CTBOX_KEY_Auto AND CTBOX_RS232.CTBOX_KEY_Manual THEN
				;
			END_IF
			
			IF (CTBOX_RS232.CTBOX_KEY_Auto AND CTBOX_RS232.CTBOX_KEY_Manual=FALSE) OR CTBOX_RS232.CTBOX_KEY_Manual AND CTBOX_RS232.CTBOX_KEY_Auto=FALSE THEN
				Step_CBCT:=60;
			END_IF
			
		60://7和8灯关闭 
			GVL_State.bEnable_CTBOX:=TRUE;
			LampCmd7:=E_LampCmd.关闭;
			LampCmd8:=E_LampCmd.关闭;
			WorkStation_TCP.PLC_SEND1.m_nFocus:=0;	//关闭按键提示0228
			TON_C60(IN:= TRUE, PT:=T#1S , Q=> , ET=> );
			
			IF TON_C60.Q THEN
				Step_CBCT:=70;
			END_IF
			
		70://扫描中间态，给跳转用的
			GVL_State.bEnable_CTBOX:=FALSE;//关闭CTBOX发送灯使能
			WorkStation_TCP.PLC_SEND1.m_nMoveState	:=1;	//send[9]
			WorkStation_TCP.PLC_SEND1.m_nScanProType:=2;	//send[16]
			TON_C70(IN:=TRUE , PT:=T#2S , Q=> , ET=> );
			TON_C220(IN:=FALSE);TON_C72(IN:=FALSE);
			Axis_QJ.QJ_AxisCmd.bAbs:=FALSE;//复位前进轴
			Axis_XZ.XZ_AxisCmd.bAbs:=FALSE;//复位旋转轴
			TON_C72(IN:=FALSE);
			TON_C79(IN:=TRUE , PT:= T#1S, Q=> , ET=> );
			
			IF XRAY_RS485.Standby_Step=60 THEN  //保证写入参数
				Entity_IO.bXaryOne:=TRUE;//开启透视
			END_IF;
			
			(*判断是否最后一次扫描*)
			IF WorkStation_TCP.PLC_RECV1.m_nLastMsg=1 THEN
				bCBCTLast := TRUE;
			ELSE
				bCBCTLast := FALSE;
			END_IF
			
			(*跳转指令*)
			IF TON_C70.Q AND Entity_IO.bXaryOne THEN
				Step_CBCT:=79;
			END_IF
			
		74:
			Entity_IO.bXaryOne:=FALSE;
			GVL_SCAN.bJumpScan:=TRUE;		//结束扫描，射线源超时报警了，EL019，结束扫描
			Step_CBCT:=74;
			
		79:
			Axis_XZ.XZ_AxisCmd.bAbs:=FALSE;
			TON_C80_ABS(IN:=FALSE);
			TON_C79(IN:=TRUE , PT:= T#4S, Q=> , ET=> );
			IF TON_C79.Q THEN
				Step_CBCT:=80;
			END_IF
			
		80://第一次自动扫描
			(*1.给上位机发送的数*)
			TON_C79(IN:=FALSE);
			WorkStation_TCP.PLC_SEND1.m_nMoveState	:=2;
			WorkStation_TCP.PLC_SEND1.m_nScanProType:=2;

			(*2.触发旋转轴运动*)
			Axis_XZ.XZ_AxisCmd.AxisPara.rAbsPosition:=LIMIT(-3,WorkStation_TCP.PLC_RECV1.m_nRotateEnd,363);
			Axis_XZ.XZ_AxisCmd.AxisPara.rAbsVelocity:=XZ_Velocity;
			TON_C80_ABS(IN:=TRUE , PT:=T#1S );
			Axis_XZ.XZ_AxisCmd.bAbs:=TON_C80_ABS.Q;
					
			(*4.开启允许曝光指令*)
			IF Entity_IO.bXaryOne AND (Axis_XZ.XZ_AxisState.rActPosition>=MIN(WorkStation_TCP.PLC_RECV1.m_nAngleStart,WorkStation_TCP.PLC_RECV1.m_nAngleEnd)) 
				AND (Axis_XZ.XZ_AxisState.rActPosition<=MAX(WorkStation_TCP.PLC_RECV1.m_nAngleStart,WorkStation_TCP.PLC_RECV1.m_nAngleEnd))  THEN
				GVL_SCAN.bEnableTrigger:=TRUE;
			ELSE
				GVL_SCAN.bEnableTrigger:=FALSE;
			END_IF 
			
			(*5.跳转,到达终止角度*)
			TON_C80(IN:= ABS(Axis_XZ.XZ_AxisState.rActPosition-WorkStation_TCP.PLC_RECV1.m_nRotateEnd)<1, PT:=T#2S , Q=> , ET=> );	
			IF TON_C80.Q THEN
				Step_CBCT:=81;
			END_IF
			
			(*6.透视信号超时报警，射线源30秒连续开启曝光会报警*)
			TON_C72(IN:=Entity_IO.bXaryOne , PT:=T#5M , Q=> , ET=> );
			IF TON_C72.Q THEN
				Step_CBCT:=74;	
			END_IF
			
		81://出射线状态结束，采集射线源状态机信息
			Entity_IO.bXaryOne		:=FALSE;
			TON_C90(IN:=FALSE , PT:=T#2S , Q=> , ET=> );
			IF XRAY_RS485.Main_Step=20 THEN
				Step_CBCT:=90;
			END_IF
			
		90://中间变量清零1070
			Axis_XZ.XZ_AxisCmd.bAbs	:=FALSE;	
			Entity_IO.bXaryOne		:=FALSE;
			TON_C100(IN:= FALSE, PT:=T#2S);
			C_100:=FALSE;
			WorkStation_TCP.PLC_SEND1.m_nMoveState:=3; //send [9]
			TON_C90(IN:=TRUE , PT:=T#2S , Q=> , ET=> );
			IF TON_C90.Q THEN
				IF (WorkStation_TCP.PLC_RECV1.m_nCircleIndex+1)>=(WorkStation_TCP.PLC_RECV1.m_nCircleCount) AND bCBCTLast THEN //最后一次扫描退出
					GVL_SCAN.bJumpScan:=TRUE;
				END_IF
			END_IF
			
			C_100:=FALSE;
			TON_C80_ABS(IN:=FALSE);
			
			(*增加跳转判断*)
			IF WorkStation_TCP.PLC_RECV1.m_nSocketType=1 THEN 	//增加第二次运动判断，m_nSocketType=1 
				Step_CBCT:=100;
			END_IF
			
		100:	
			C_100:=TRUE;
			(*延迟2秒*)
			TON_C100(IN:= C_100, PT:=T#1S);
			(*跳转*)
			IF TON_C100.Q THEN
				Step_CBCT:=110;
			END_IF;
			
		110://CBCT下的自动扫还是手动扫，根据上位机命令
			TON_C210(IN:= FALSE);TON_C201(IN:=FALSE);
			C_100:=FALSE;
			
			IF WorkStation_TCP.PLC_RECV1.m_nScanUseType=1 THEN
				Step_CBCT:=200;		//手动扫描
			ELSE
				Step_CBCT:=120;		//自动扫描
			END_IF
		 
		120://开启自动扫描
			TOF_C80(IN:= FALSE);TON_C100(IN:=FALSE);TON_C90(IN:=FALSE);TON_C80(IN:=FALSE);TON_C70(IN:=FALSE);TON_C60(IN:=FALSE);
			Axis_QJ.QJ_AxisCmd.AxisPara.rAbsPosition:=LIMIT(0,WorkStation_TCP.PLC_RECV1.m_fScanTop,900);
			Axis_QJ.QJ_AxisCmd.bAbs:=TRUE;
			
			IF ABS(Axis_QJ.QJ_AxisState.rActPosition-Axis_QJ.QJ_AxisCmd.AxisPara.rAbsPosition)<1 THEN
				WorkStation_TCP.PLC_SEND1.m_nMoveState:=1; 			//send [9]
				Step_CBCT:=70;				//自动扫描
			ELSE
				WorkStation_TCP.PLC_SEND1.m_nMoveState:=0; 			//send [9]	//0-准备过程中 1-准备完成 2-曝光中 3-本次扫描结束
			END_IF
			
		(*-------------------------手动扫描-----------------------------*)	
		200://中间状态清零
			WorkStation_TCP.PLC_SEND1.m_nMoveState:=0; //send [9]	//0-准备过程中 1-准备完成 2-曝光中 3-本次扫描结束
			Axis_XZ.XZ_AxisCmd.bAbs:=FALSE;
			Step_CBCT:=201;

		201:
			TON_C201(IN:= TRUE, PT:=T#1S , Q=> , ET=> );
			IF TON_C201.Q THEN
				Step_CBCT:=210;
			END_IF
			
		210://7灯闪烁，机架运动到目标位置
			(*1.发送给上位机的数据*)
			WorkStation_TCP.PLC_SEND1.m_nMoveState:=0; //send [9]	//0-准备过程中 1-准备完成 2-曝光中 3-本次扫描结束
			TON_C201(IN:= FALSE);
			(*2.7灯闪烁*)
			GVL_State.bEnable_CTBOX:=TRUE;			//开启CTBOX发送灯使能
			LampCmd7:=E_LampCmd.慢闪;
			WorkStation_TCP.PLC_SEND1.m_nFocus:=7;	//按键提示0228
			
			(*3.旋转轴运动到目标位置*)
			Axis_XZ.XZ_AxisCmd.AxisPara.rAbsPosition:=LIMIT(-4,WorkStation_TCP.PLC_RECV1.m_nRotateBegin,363);
			Axis_XZ.XZ_AxisCmd.AxisPara.rAbsVelocity:=XZ_Velocity;
			
			IF WorkStation_TCP.PLC_RECV1.m_nSocketType=1 THEN
				Axis_XZ.XZ_AxisCmd.bAbs:=TRUE;
			END_IF;
			
			(*4.到位后2秒跳转*)
			TON_C210(IN:=ABS(Axis_XZ.XZ_AxisState.rActPosition-WorkStation_TCP.PLC_RECV1.m_nRotateBegin)<1 , PT:=T#1S , Q=> , ET=> );
			IF TON_C210.Q THEN
				Step_CBCT:=221;	
			END_IF
		
		221://中间状态清零
			Axis_XZ.XZ_AxisCmd.bAbs:=FALSE;
			Axis_QJ.QJ_AxisCmd.bAbs:=FALSE;
			GVL_State.bEnable_CTBOX:=FALSE;//关闭CTBOX发送灯使能
			Step_CBCT:=220;
			
		220://用户按7键，床自动走到预设位置
			(*1.按7键关闭7灯*)
			IF CTBOX_RS232.CTBOX_KEY_Manual THEN
				LampCmd7:=E_LampCmd.关闭;
				GVL_State.bEnable_CTBOX:=TRUE;//开启CTBOX发送灯使能
				WorkStation_TCP.PLC_SEND1.m_nFocus:=0;	//关闭按键提示0228
			END_IF
			
			(*2.触发床运动*)
			R_TRIG_C220(CLK:=CTBOX_RS232.CTBOX_KEY_Manual , Q=> );
			Axis_QJ.QJ_AxisCmd.AxisPara.rAbsPosition:=LIMIT(0,WorkStation_TCP.PLC_RECV1.m_fScanTop,900);
			Axis_QJ.QJ_AxisCmd.bAbs:=R_TRIG_C220.Q;
			
			(*3.跳转指令*)
			IF ABS(Axis_QJ.QJ_AxisState.rActPosition-WorkStation_TCP.PLC_RECV1.m_fScanTop)<1 AND (LampCmd7=E_LampCmd.关闭) THEN //保证必须按下7键
				WorkStation_TCP.PLC_SEND1.m_nMoveState:=1; //send [9]	//0-准备过程中 1-准备完成 2-曝光中 3-本次扫描结束
			ELSE
				WorkStation_TCP.PLC_SEND1.m_nMoveState:=0; //send [9]	//0-准备过程中 1-准备完成 2-曝光中 3-本次扫描结束
			END_IF
			
			(*4.延迟跳转，保证send [9]发送*)
			TOF_C80(IN:= FALSE);TON_C100(IN:=FALSE);TON_C90(IN:=FALSE);TON_C80(IN:=FALSE);TON_C70(IN:=FALSE);TON_C60(IN:=FALSE);
			TON_C210(IN:=FALSE);TON_C72(IN:=FALSE);TON_C201(IN:=FALSE);
			TON_C220(IN:=(WorkStation_TCP.PLC_SEND1.m_nMoveState=1) , PT:=T#2S , Q=> , ET=> );
			IF TON_C220.Q THEN
				Step_CBCT:=70;
			END_IF		
	END_CASE
END_ACTION

ACTION _a_Homing_active:

(*回零*)
	TON_Home(IN:= TRUE, PT:= T#5S, Q=> , ET=> );

	Axis_XZ.XZ_AxisCmd.AxisPara.rSetPosition:=0;
	Axis_XZ.XZ_AxisCmd.bHome:=TON_Home.Q;

	Axis_QJ.QJ_AxisCmd.AxisPara.rSetPosition:=0;
	Axis_QJ.QJ_AxisCmd.bHome:=TON_Home.Q;
	
(*5.1 回零参数*)
(*	fbMC_HomePara(	Axis:= ASDA_A3_Drive_XZ, 
					Exec:= XZ_AxisCmd.bSetHomePara, 
					HomeMode:=XZ_AxisCmd.AxisPara.iHomeMode , 
					HomeHighSpeed:=dHomeHighSpeed , 
					HomeLowSpeed:= dHomeLowSpeed , 
					Acceleration:= dHomeAcc , 
					Done=> , 
					Busy=> , 
					Error=> , 
					Error_CANopenKenel=> , 
					Error_SDO=> );
*)					
(*5.2 执行回零命令*)
//	fbMC_Home(Axis:=  ASDA_A3_Drive_XZ, Execute:=XZ_AxisCmd.bHome , Position:=dSetPosition);

	LampCmd5:=E_LampCmd.关闭;
	LampCmd6:=E_LampCmd.关闭;
	LampCmd7:=E_LampCmd.关闭;
	LampCmd8:=E_LampCmd.关闭;

	IF (Axis_QJ.fbMC_Home.Done AND Axis_XZ.fbMC_Home.Done) THEN
		bHomingDone:=TRUE;
	ELSE
		bHomingDone:=FALSE;	
	END_IF
END_ACTION

TRANSITION T_MoveXZ:

(*进入旋转轴运动模式*)
	WorkStation_TCP.PLC_RECV1.m_nSocketType=1 AND WorkStation_TCP.PLC_RECV1.m_nExpId=5
END_TRANSITION

ACTION _a_SelfCheck_entry:

	Axis_XZ.XZ_AxisCmd.bPower:=TRUE;//上使能
	Axis_QJ.QJ_AxisCmd.bPower:=TRUE;//上使能
	Entity_IO.bBrakeOut:=TRUE;//打开抱闸
END_ACTION

ACTION _a_MoveXZ_exit:


	LampCmd5:=E_LampCmd.关闭;
	LampCmd6:=E_LampCmd.关闭;
	LampCmd7:=E_LampCmd.关闭;
	LampCmd8:=E_LampCmd.关闭;
	
	Entity_IO.bTriggerPannel:=FALSE;
	Entity_IO.bTriggerOut:=FALSE;

	TON_S30(IN:= FALSE );
END_ACTION

TRANSITION T_CBCT:


(*进入CBCT扫描*)
	WorkStation_TCP.PLC_RECV1.m_nSocketType=1 AND WorkStation_TCP.PLC_RECV1.m_nExpId=2
END_TRANSITION

ACTION _a_Emergercy_entry:

GVL_State.iPLC_State:=70;
END_ACTION

ACTION _AutoDR_entry_0:


GVL_State.iPLC_State:=58;
Step_AutoDR:=0; 
GVL_SCAN.bJumpScan:=FALSE;
bTCP_Socket:=TRUE;

GVL_SCAN.bEnableScout:=FALSE;
GVL_SCAN.bEnableTrigger:=FALSE;
END_ACTION

ACTION _a_ScoutScan_entry:


Step_Scout:=0; 

GVL_State.iPLC_State:=50;

bTCP_Socket:=TRUE; //首次开机需要按2下开始采集
END_ACTION

ACTION _a_ScoutScan_exit:



	LampCmd5:=E_LampCmd.关闭;
	LampCmd6:=E_LampCmd.关闭;
	LampCmd7:=E_LampCmd.关闭;
	LampCmd8:=E_LampCmd.关闭;
	
	GVL_SCAN.bEnableScout:=FALSE;
	
	Entity_IO.bTriggerPannel:=FALSE;
	Entity_IO.bTriggerOut:=FALSE;
END_ACTION

ACTION _a_ShutDown_entry:

	(**)
	GVL_State.iPLC_State:=90;
	(*伺服电机停止*)
	Axis_XZ.XZ_AxisCmd.bStop:=TRUE;
	Axis_QJ.QJ_AxisCmd.bStop:=TRUE;
	
	(*射线停止输出*)
	Entity_IO.bXaryTwo:=FALSE;
	Entity_IO.bXaryOne:=FALSE;
	
	bOver:=FALSE;
END_ACTION

ACTION _a_Idle_active:

(*待机工作状态*)
	
	CASE Step_Idle OF
	0: //中间状态复位
		GVL_State.bEnable_CTBOX:=TRUE;	
		GVL_State.bBooting:=TRUE;
		Entity_IO.bXaryOne:=FALSE;				//试一试在这里高压会不会报错
		WorkStation_TCP.PLC_SEND1.m_nFocus:=0;	//按键提示清零0228
		TON_I00(IN:=FALSE , PT:= , Q=> , ET=> );
		TON_I10(IN:=FALSE , PT:= , Q=> , ET=> );
		TON_I20(IN:=FALSE , PT:= , Q=> , ET=> );
		TON_I30(IN:=FALSE , PT:= , Q=> , ET=> );
		TON_I40(IN:=FALSE , PT:= , Q=> , ET=> );
		TON_I50(IN:=FALSE , PT:= , Q=> , ET=> );
		TON_IDLE(IN:=FALSE, PT:= , Q=> , ET=> );
		Step_Idle:=10;
		
	10:	//所有运动立刻停止，所有灯关闭
		TON_I00(IN:=TRUE , PT:=T#1S , Q=> , ET=> );
		TON_I10(IN:=TRUE , PT:=T#1S , Q=> , ET=> );
		Axis_QJ.QJ_AxisCmd.bStop:=TON_I00.Q;
		Axis_XZ.XZ_AxisCmd.bStop:=TON_I10.Q;
		
		LampCmd5:=E_LampCmd.关闭;
		LampCmd6:=E_LampCmd.关闭;
		LampCmd7:=E_LampCmd.关闭;
		LampCmd8:=E_LampCmd.关闭;
		
		TON_IDLE(IN:= TRUE, PT:=T#2S , Q=> , ET=> );
		IF TON_IDLE.Q THEN
			Step_Idle:=20;
		END_IF
		
	20:	//中间变量复位
		Axis_QJ.QJ_AxisCmd.bStop:=FALSE;
		Axis_XZ.XZ_AxisCmd.bStop:=FALSE;
		TON_IDLE(IN:= FALSE, PT:=T#2S , Q=> , ET=> );
		Step_Idle:=30;
		
	30:	//待机模式准备，开启点动运动权限
		GVL_State.iPLC_State:=40;
		(*0.给射线源写入参数的一个标志位0214*)
		GVL_State.bBooting:=FALSE;
		(*1.给上位机发送数据*)
		WorkStation_TCP.PLC_SEND1.m_nExpStates	:=1;//[4]为曝光状态，枚举值，0:idle（空闲） 1:prep（训机） 2: ready（训机结束，准备完成，可以出束） 3: XrayOn（出射线） 4:XrayOff（关射线） 5 error；
		WorkStation_TCP.PLC_SEND1.m_nMoveState	:=0;//[9]起始、终止状态， 默认值-1， 0为当前扫描方案处于准备好状态，可以准备扫描；1为当前扫描方案结束，运动过程中值为-1
		WorkStation_TCP.PLC_SEND1.m_nScanProType:=2;//[16]执行扫描方案的类型，0为自动扫描，1为手动扫描，2为无设置意义的值，默认值为2
		
		(*2.开启前进轴和升降轴运动*)
		(*2.1 升降轴运动*)
		Motor_SJ(Enable:= TRUE);
		
		(*2.2 前进轴控制*)
		(*2.1 相对运动*)
		Axis_QJ.QJ_AxisCmd.AxisPara.rRelVelocity:=80;
		Axis_QJ.QJ_AxisCmd.AxisPara.rRelPosition:=50;
		IF Axis_QJ.QJ_AxisState.rActPosition<=900 THEN
			Axis_QJ.QJ_AxisCmd.bRel:=Entity_IO.LeftPannel_DistanceMove OR Entity_IO.RightPannel_DistanceMove;
		ELSE
			Axis_QJ.QJ_AxisCmd.bRel:=FALSE;
		END_IF
		
		(*2.2 点动和绝对运动合并程序*)
		Axis_QJ.QJ_AxisCmd.AxisPara.rAbsVelocity:=80;
		(*2.2.1 点动触发逻辑*)
		R_TRIG_Jog(CLK:= (Entity_IO.LeftPannel_BedFore OR Entity_IO.RightPannel_BedFore OR CTBOX_RS232.CTBOX_KEY_BedFore)
					OR (Entity_IO.LeftPannel_BedBack OR Entity_IO.RightPannel_BedBack OR CTBOX_RS232.CTBOX_KEY_BedBack), Q=> ); //获取上升沿
		F_TRIG_Jog(CLK:= (Entity_IO.LeftPannel_BedFore OR Entity_IO.RightPannel_BedFore OR CTBOX_RS232.CTBOX_KEY_BedFore)
					OR (Entity_IO.LeftPannel_BedBack OR Entity_IO.RightPannel_BedBack OR CTBOX_RS232.CTBOX_KEY_BedBack), Q=> ); //获取上升沿

		(*2.2.2 点动最大最小位置，绝对运动走记录值*)
		IF Entity_IO.LeftPannel_BedFore OR Entity_IO.RightPannel_BedFore OR CTBOX_RS232.CTBOX_KEY_BedFore THEN
			Axis_QJ.QJ_AxisCmd.AxisPara.rAbsPosition:=900;
		ELSE
			IF Entity_IO.LeftPannel_BedBack OR Entity_IO.RightPannel_BedBack OR CTBOX_RS232.CTBOX_KEY_BedBack THEN
				Axis_QJ.QJ_AxisCmd.AxisPara.rAbsPosition:=0;
			ELSE
				Axis_QJ.QJ_AxisCmd.AxisPara.rAbsPosition:=LIMIT(0,rBedRecordLength,900); 
			END_IF
		END_IF
		
		(*2.2.3 触发绝对运动，按键或者触发走记录位置*)
		Axis_QJ.QJ_AxisCmd.bAbs	:=R_TRIG_Jog.Q OR  Entity_IO.LeftPannel_MoveRecordPos OR Entity_IO.RightPannel_MoveRecordPos;
		
		(*2.2.4 触发停止*)
		R_RelStop(CLK:= (Axis_QJ.QJ_AxisState.rActPosition>901), Q=> ); 
		Axis_QJ.QJ_AxisCmd.bStop:=F_TRIG_Jog.Q OR R_RelStop.Q;
		
	END_CASE
		
	
	
	(*	Axis_QJ.QJ_AxisCmd.AxisPara.rAbsVelocity:=80;

		R_TRIG_Jog(CLK:= (Entity_IO.LeftPannel_BedFore OR Entity_IO.RightPannel_BedFore OR CTBOX_RS232.CTBOX_KEY_BedFore)
					OR (Entity_IO.LeftPannel_BedBack OR Entity_IO.RightPannel_BedBack OR CTBOX_RS232.CTBOX_KEY_BedBack), Q=> ); //获取上升沿
		F_TRIG_Jog(CLK:= (Entity_IO.LeftPannel_BedFore OR Entity_IO.RightPannel_BedFore OR CTBOX_RS232.CTBOX_KEY_BedFore)
					OR (Entity_IO.LeftPannel_BedBack OR Entity_IO.RightPannel_BedBack OR CTBOX_RS232.CTBOX_KEY_BedBack), Q=> ); //获取上升沿

		(*启动运动*)
		IF Entity_IO.LeftPannel_BedFore OR Entity_IO.RightPannel_BedFore OR CTBOX_RS232.CTBOX_KEY_BedFore THEN
			Axis_QJ.QJ_AxisCmd.AxisPara.rAbsPosition:=900;
		ELSE
			IF Entity_IO.LeftPannel_BedBack OR Entity_IO.RightPannel_BedBack OR CTBOX_RS232.CTBOX_KEY_BedBack THEN
				Axis_QJ.QJ_AxisCmd.AxisPara.rAbsPosition:=0;
			ELSE
				Axis_QJ.QJ_AxisCmd.AxisPara.rAbsPosition:=Axis_QJ.QJ_AxisCmd.AxisPara.rAbsPosition;
			END_IF
		END_IF

		Axis_QJ.QJ_AxisCmd.bAbs	:=R_TRIG_Jog.Q;
		(*触发停止*)
		Axis_QJ.QJ_AxisCmd.bStop:=F_TRIG_Jog.Q;
		
		(*2.2 升降轴控制，已集成到子程序里了*)
		Motor_SJ(Enable:= TRUE);
		
		(*2.2 补充位置控制，当Pannel面板操作记录预设位置时，升降轴和前进轴，自动走到预设位置*)
		IF Entity_IO.LeftPannel_MoveRecordPos OR Entity_IO.RightPannel_MoveRecordPos THEN
			Axis_QJ.QJ_AxisCmd.AxisPara.rAbsPosition:=LIMIT(0,rBedRecordLength,900);
			R_MoveRecordPos(CLK:= (Entity_IO.LeftPannel_MoveRecordPos OR Entity_IO.RightPannel_MoveRecordPos), Q=> );	
			Axis_QJ.QJ_AxisCmd.bAbs:=R_MoveRecordPos.Q;
		ELSE
			;
		END_IF;	
		;
		
		(*2.3 绝对运动*)
		Axis_QJ.QJ_AxisCmd.AxisPara.rAbsVelocity:=80;
		Axis_QJ.QJ_AxisCmd.AxisPara.rAbsPosition:=LIMIT(0,rBedRecordLength,900);
		Axis_QJ.QJ_AxisCmd.bAbs:= Entity_IO.LeftPannel_MoveRecordPos OR Entity_IO.RightPannel_MoveRecordPos;
		
		
		(*2.1 点动*)
		Axis_QJ.QJ_AxisCmd.AxisPara.rJogVelocity:=80;
		IF Axis_QJ.QJ_AxisState.rActPosition<=850 THEN
			Axis_QJ.QJ_AxisCmd.bJogP:=Entity_IO.LeftPannel_BedFore OR Entity_IO.RightPannel_BedFore OR CTBOX_RS232.CTBOX_KEY_BedFore;
		ELSE
			Axis_QJ.QJ_AxisCmd.bJogP:=FALSE;
		END_IF
		
		IF Axis_QJ.QJ_AxisState.rActPosition>=80 THEN
			Axis_QJ.QJ_AxisCmd.bJogN:=Entity_IO.LeftPannel_BedBack OR Entity_IO.RightPannel_BedBack OR CTBOX_RS232.CTBOX_KEY_BedBack;
		ELSE
			Axis_QJ.QJ_AxisCmd.bJogN:=FALSE;
		END_IF;
	*)
END_ACTION

ACTION _a_Error_exit:


		Axis_QJ.QJ_AxisCmd.bReset:=FALSE;
		Axis_XZ.XZ_AxisCmd.bReset:=FALSE;
END_ACTION

ACTION _a_ShutDown_active:

(*关机模式*)

(*1.伺服电机下使能*)
	Axis_XZ.XZ_AxisCmd.bPower:=FALSE;
	Axis_QJ.QJ_AxisCmd.bPower:=FALSE;
	
	Entity_IO.bBrakeOut:=FALSE;//
	
(*2.运动都停止*)
	Axis_XZ.XZ_AxisCmd.bStop:=FALSE;
	Axis_QJ.QJ_AxisCmd.bStop:=FALSE;
	
	Motor_SJ(Enable:= FALSE);

(*3.无法出束，控制二档信号*)
	Entity_IO.bXaryTwo:=FALSE;
	Entity_IO.bXaryOne:=FALSE;
	
(*4.记录参数*)
END_ACTION

ACTION _a_Homing_entry:

	GVL_State.iPLC_State:=30;
	
	Axis_QJ.QJ_AxisCmd.bSetHomePara:=FALSE;
	Axis_XZ.XZ_AxisCmd.bSetHomePara:=FALSE;
	
	bHomingDone:=FALSE;
	
	Axis_XZ.XZ_AxisCmd.bHome:=FALSE;
	Axis_QJ.QJ_AxisCmd.bHome:=FALSE;
	
	TON_Home(IN:= FALSE);
END_ACTION

ACTION _a_CBCTScan_entry:

GVL_State.iPLC_State:=60;
Step_CBCT:=0; 
GVL_SCAN.bJumpScan:=FALSE;
bTCP_Socket:=TRUE;

GVL_SCAN.bEnableScout:=FALSE;
GVL_SCAN.bEnableTrigger:=FALSE;

GVL_State.bEnable_CTBOX:=FALSE;//进入使能CTBOX——Enable
END_ACTION

ACTION _a_QuickScan_active:

	CASE Step_QuickScan OF 
		0:	//初始化准备流程
			(*1.给上位机发送的数据*)
			WorkStation_TCP.PLC_SEND1.m_nMoveState:=0;			//send[9] //0-准备过程中 1-准备完成 2-曝光中 3-本次扫描结束
			bTCP_Socket:=FALSE; 
			bCBCTLast:=FALSE;
			
			(*2.运动准备数据*)
			(*2.1 写入旋转速度参数*)
			IF WorkStation_TCP.PLC_RECV1.m_fSecondPerCicle<>0 THEN//避免除零
				Axis_XZ.XZ_AxisCmd.AxisPara.rAbsVelocity:=UDINT_TO_REAL(LIMIT(360/300 ,360/WorkStation_TCP.PLC_RECV1.m_fSecondPerCicle ,360/8 ));		//修改最快速度360/20 0613
				XZ_Velocity:=LIMIT(360/300 ,360/UDINT_TO_REAL(WorkStation_TCP.PLC_RECV1.m_fSecondPerCicle) ,360/8);
			ELSE
				Axis_XZ.XZ_AxisCmd.AxisPara.rAbsVelocity:=8;
			END_IF;
			GVL_State.bEnable_CTBOX:=FALSE;//关闭CTBOX发送灯使能
			Step_QuickScan:=10;

		10:	//运动过程中变量复位标志
			TON_C20(IN:= FALSE);TON_C30(IN:= FALSE);
			TON_C40(IN:= FALSE);TON_C50(IN:= FALSE);TON_C60(IN:= FALSE);
			TON_C70(IN:= FALSE);TON_C80(IN:= FALSE);TON_C72(IN:=FALSE);
			TON_C210(IN:= FALSE);TON_C220(IN:= FALSE);TON_C230(IN:= FALSE);
			TON_C240(IN:= FALSE);TON_C250(IN:= FALSE);
			TON_C20_ABS(IN:=FALSE);
			TOF_C80(IN:= FALSE);
			Axis_XZ.XZ_AxisCmd.bAbs:=FALSE;
			Step_QuickScan:=20;
			
		20://按5键，移动床到预设位置，松开即停，机架直接到预设位置
			(*1.发送给上位机的数据*)
			WorkStation_TCP.PLC_SEND1.m_nExpStates:=1;		//0-准备过程中 1-准备完成 2-曝光中 3-本次扫描结束	
			WorkStation_TCP.PLC_SEND1.m_nMoveState:=0;		//起始、终止状态， 默认值0， 1为当前扫描方案处于准备好状态，可以准备扫描；2为当前扫描方案结束，运动过程中值为0
			WorkStation_TCP.PLC_SEND1.m_nScanProType:=2;	//扫描方案类型 , 1-手动，0-自动. 
			
			(*2.旋转轴直接运动到目标位置*)
			Axis_XZ.XZ_AxisCmd.AxisPara.rAbsPosition:=LIMIT(-3,WorkStation_TCP.PLC_RECV1.m_nRotateBegin,363);
			Axis_XZ.XZ_AxisCmd.AxisPara.rAbsVelocity:=18;
			TON_C20_ABS(IN:=TRUE , PT:=T#1S);
			Axis_XZ.XZ_AxisCmd.bAbs:=TON_C20_ABS.Q;
			
			(*3.前进轴运动*)
			R_TRIG_C20(CLK:= CTBOX_RS232.CTBOX_KEY_MoveDistance, Q=> );//触发运动
			F_TRIG_C20(CLK:= CTBOX_RS232.CTBOX_KEY_MoveDistance, Q=> );//触发停止
			
			Axis_QJ.QJ_AxisCmd.bAbs	:=R_TRIG_C20.Q;
			Axis_QJ.QJ_AxisCmd.AxisPara.rAbsPosition	:=LIMIT(0,WorkStation_TCP.PLC_RECV1.m_fScanTop,900);
			Axis_QJ.QJ_AxisCmd.bStop:=F_TRIG_C20.Q;
			
			(*4.5灯逻辑处理*)
			GVL_State.bEnable_CTBOX:=TRUE;//开启CTBOX发送灯使能
			IF ABS(Axis_QJ.QJ_AxisState.rActPosition-WorkStation_TCP.PLC_RECV1.m_fScanTop)>1 THEN
				LampCmd5:=E_LampCmd.慢闪;
				WorkStation_TCP.PLC_SEND1.m_nFocus:=5;//按键提示0228
			ELSE
				LampCmd5:=E_LampCmd.关闭;
				WorkStation_TCP.PLC_SEND1.m_nFocus:=0;//关闭按键提示0228
			END_IF
			
			(*5.跳转*)
			TON_C20(IN:=ABS(Axis_QJ.QJ_AxisState.rActPosition-WorkStation_TCP.PLC_RECV1.m_fScanTop)<1 
				AND ABS(Axis_XZ.XZ_AxisState.rActPosition-WorkStation_TCP.PLC_RECV1.m_nRotateBegin)<1 , PT:=T#2S);
			IF TON_C20.Q THEN  
				Step_QuickScan:=30;
			END_IF
			
		30:	//射线源参数写入成功标志
			TON_C20_ABS(IN:=FALSE);
			LampCmd5:=E_LampCmd.关闭;
			Axis_XZ.XZ_AxisCmd.bAbs:=FALSE;
			Axis_QJ.QJ_AxisCmd.bAbs:=FALSE;
			Axis_QJ.QJ_AxisCmd.bStop:=FALSE;
			IF XRAY_RS485.Standby_Step=60 THEN      //这里需要修改 0610未修改
				Step_QuickScan:=40;
			END_IF
			
		40:	//7灯和8灯开始慢闪
			WorkStation_TCP.PLC_SEND1.m_nMoveState:=1;		//起始、终止状态， 默认值0， 1为当前扫描方案处于准备好状态
			LampCmd7:=E_LampCmd.慢闪;
			LampCmd8:=E_LampCmd.慢闪;
			WorkStation_TCP.PLC_SEND1.m_nFocus:=8;//按键提示0228
			TON_C40(IN:=TRUE , PT:=T#600MS , Q=> , ET=> );
			IF TON_C40.Q THEN
				Step_QuickScan:=41;
			END_IF
		41:
			GVL_State.bEnable_CTBOX:=FALSE;//开启CTBOX发送灯使能
			Step_QuickScan:=50;
			
		50://用户选择自动扫描或手动扫描
			IF CTBOX_RS232.CTBOX_KEY_Auto=FALSE AND CTBOX_RS232.CTBOX_KEY_Manual THEN
				WorkStation_TCP.PLC_SEND1.m_nScanProType:=1;								//扫描方案类型 , 1-手动，0-自动. 
				bCBCT_AUTO_Manual:=TRUE;
			ELSIF CTBOX_RS232.CTBOX_KEY_Auto AND CTBOX_RS232.CTBOX_KEY_Manual=FALSE THEN
				WorkStation_TCP.PLC_SEND1.m_nScanProType:=0;								//扫描方案类型 , 1-手动，0-自动. 
				bCBCT_AUTO_Manual:=FALSE;
			ELSIF CTBOX_RS232.CTBOX_KEY_Auto=FALSE AND CTBOX_RS232.CTBOX_KEY_Manual=FALSE THEN
				;
			ELSIF CTBOX_RS232.CTBOX_KEY_Auto AND CTBOX_RS232.CTBOX_KEY_Manual THEN
				;
			END_IF
			
			IF (CTBOX_RS232.CTBOX_KEY_Auto AND CTBOX_RS232.CTBOX_KEY_Manual=FALSE) OR CTBOX_RS232.CTBOX_KEY_Manual AND CTBOX_RS232.CTBOX_KEY_Auto=FALSE THEN
				Step_QuickScan:=60;
			END_IF
			
		60://7和8灯关闭 
			GVL_State.bEnable_CTBOX:=TRUE;
			LampCmd7:=E_LampCmd.关闭;
			LampCmd8:=E_LampCmd.关闭;
			WorkStation_TCP.PLC_SEND1.m_nFocus:=0;	//关闭按键提示0228
			TON_C60(IN:= TRUE, PT:=T#1S , Q=> , ET=> );
			
			IF TON_C60.Q THEN
				Step_QuickScan:=70;
			END_IF
			
		70://扫描中间态，给跳转用的
			GVL_State.bEnable_CTBOX:=FALSE;//关闭CTBOX发送灯使能
			WorkStation_TCP.PLC_SEND1.m_nMoveState	:=1;	//send[9]
			WorkStation_TCP.PLC_SEND1.m_nScanProType:=2;	//send[16]
			TON_C70(IN:=TRUE , PT:=T#2S , Q=> , ET=> );
			TON_C220(IN:=FALSE);TON_C72(IN:=FALSE);
			Axis_QJ.QJ_AxisCmd.bAbs:=FALSE;//复位前进轴
			Axis_XZ.XZ_AxisCmd.bAbs:=FALSE;//复位旋转轴
			TON_C72(IN:=FALSE);
			TON_C79(IN:=TRUE , PT:= T#1S, Q=> , ET=> );
			
			IF XRAY_RS485.Standby_Step=60 THEN  //保证写入参数
				Entity_IO.bXaryOne:=TRUE;		//开启透视
			END_IF;
			
			(*判断是否最后一次扫描*)
			IF WorkStation_TCP.PLC_RECV1.m_nLastMsg=1 THEN
				bCBCTLast := TRUE;
			ELSE
				bCBCTLast := FALSE;
			END_IF
			
			(*跳转指令*)
			IF TON_C70.Q AND Entity_IO.bXaryOne THEN
				Step_QuickScan:=79;
			END_IF
			
		74:
			Entity_IO.bXaryOne:=FALSE;
			GVL_SCAN.bJumpScan:=TRUE;		//结束扫描，射线源超时报警了，EL019，结束扫描
			Step_QuickScan:=74;
			
		79:
			Axis_XZ.XZ_AxisCmd.bAbs:=FALSE;
			TON_C80_ABS(IN:=FALSE);
			TON_C79(IN:=TRUE , PT:= T#1S, Q=> , ET=> );			//连续透视模式，这个时间减小，之前4秒0611
			IF TON_C79.Q THEN
				Step_QuickScan:=80;
			END_IF
			
		80://第一次自动扫描			//还得告诉上位机什么时候开始内触发，什么时候结束，可以根据射线源状态=30的时候开始内触发，Entity_IO.bXaryOne		:=FALSE;结束  PLC_SEND1.m_nDirectionState可以用这个传输
			(*1.给上位机发送的数*)
			TON_C79(IN:=FALSE);
			WorkStation_TCP.PLC_SEND1.m_nMoveState	:=2;
			WorkStation_TCP.PLC_SEND1.m_nScanProType:=2;

			(*2.触发旋转轴运动*)
			Axis_XZ.XZ_AxisCmd.AxisPara.rAbsPosition:=LIMIT(-3,WorkStation_TCP.PLC_RECV1.m_nRotateEnd,363);
			Axis_XZ.XZ_AxisCmd.AxisPara.rAbsVelocity:=XZ_Velocity;
			TON_C80_ABS(IN:=TRUE , PT:=T#1S );
			Axis_XZ.XZ_AxisCmd.bAbs:=TON_C80_ABS.Q;
					
			(*4.开启允许曝光指令，连续透视模式，无需脉冲了*)
		(*	
			IF Entity_IO.bXaryOne AND (Axis_XZ.XZ_AxisState.rActPosition>=MIN(WorkStation_TCP.PLC_RECV1.m_nAngleStart,WorkStation_TCP.PLC_RECV1.m_nAngleEnd)) 
				AND (Axis_XZ.XZ_AxisState.rActPosition<=MAX(WorkStation_TCP.PLC_RECV1.m_nAngleStart,WorkStation_TCP.PLC_RECV1.m_nAngleEnd))  THEN
				GVL_SCAN.bEnableTrigger:=TRUE;
			ELSE
				GVL_SCAN.bEnableTrigger:=FALSE;
			END_IF 
		*)	
			(*5.跳转,到达终止角度*)
			TON_C80(IN:= ABS(Axis_XZ.XZ_AxisState.rActPosition-WorkStation_TCP.PLC_RECV1.m_nRotateEnd)<1, PT:=T#2S , Q=> , ET=> );	
			IF TON_C80.Q THEN
				Step_QuickScan:=81;
			END_IF
			
			(*6.透视信号超时报警，射线源30秒连续开启曝光会报警*)
			TON_C72(IN:=Entity_IO.bXaryOne , PT:=T#5M , Q=> , ET=> );
			IF TON_C72.Q THEN
				Step_QuickScan:=74;	
			END_IF
			
		81://出射线状态结束，采集射线源状态机信息
			Entity_IO.bXaryOne		:=FALSE;
			TON_C90(IN:=FALSE , PT:=T#2S , Q=> , ET=> );
			IF XRAY_RS485.Main_Step=20 THEN
				Step_QuickScan:=90;
			END_IF
			
		90://中间变量清零1070
			Axis_XZ.XZ_AxisCmd.bAbs	:=FALSE;	
			Entity_IO.bXaryOne		:=FALSE;
			TON_C100(IN:= FALSE, PT:=T#2S);
			C_100:=FALSE;
			WorkStation_TCP.PLC_SEND1.m_nMoveState:=3; //send [9]
			TON_C90(IN:=TRUE , PT:=T#2S , Q=> , ET=> );
			IF TON_C90.Q THEN
				IF (WorkStation_TCP.PLC_RECV1.m_nCircleIndex+1)>=(WorkStation_TCP.PLC_RECV1.m_nCircleCount) AND bCBCTLast THEN //最后一次扫描退出
					GVL_SCAN.bJumpScan:=TRUE;
				END_IF
			END_IF
			
			C_100:=FALSE;
			TON_C80_ABS(IN:=FALSE);
			
			(*增加跳转判断*)
			IF WorkStation_TCP.PLC_RECV1.m_nSocketType=1 THEN 	//增加第二次运动判断，m_nSocketType=1 
				Step_QuickScan:=100;
			END_IF
			
		100:	
			C_100:=TRUE;
			(*延迟2秒*)
			TON_C100(IN:= C_100, PT:=T#1S);
			(*跳转*)
			IF TON_C100.Q THEN
				Step_QuickScan:=110;
			END_IF;
			
		110://CBCT下的自动扫还是手动扫，根据上位机命令
			TON_C210(IN:= FALSE);TON_C201(IN:=FALSE);
			C_100:=FALSE;
			
			IF WorkStation_TCP.PLC_RECV1.m_nScanUseType=1 THEN
				Step_QuickScan:=200;		//手动扫描
			ELSE
				Step_QuickScan:=120;		//自动扫描
			END_IF
		 
		120://开启自动扫描
			TOF_C80(IN:= FALSE);TON_C100(IN:=FALSE);TON_C90(IN:=FALSE);TON_C80(IN:=FALSE);TON_C70(IN:=FALSE);TON_C60(IN:=FALSE);
			Axis_QJ.QJ_AxisCmd.AxisPara.rAbsPosition:=LIMIT(0,WorkStation_TCP.PLC_RECV1.m_fScanTop,900);
			Axis_QJ.QJ_AxisCmd.bAbs:=TRUE;
			
			IF ABS(Axis_QJ.QJ_AxisState.rActPosition-Axis_QJ.QJ_AxisCmd.AxisPara.rAbsPosition)<1 THEN
				WorkStation_TCP.PLC_SEND1.m_nMoveState:=1; 			//send [9]
				Step_QuickScan:=70;				//自动扫描
			ELSE
				WorkStation_TCP.PLC_SEND1.m_nMoveState:=0; 			//send [9]	//0-准备过程中 1-准备完成 2-曝光中 3-本次扫描结束
			END_IF
			
		(*-------------------------手动扫描-----------------------------*)	
		200://中间状态清零
			WorkStation_TCP.PLC_SEND1.m_nMoveState:=0; //send [9]	//0-准备过程中 1-准备完成 2-曝光中 3-本次扫描结束
			Axis_XZ.XZ_AxisCmd.bAbs:=FALSE;
			Step_QuickScan:=201;

		201:
			TON_C201(IN:= TRUE, PT:=T#1S , Q=> , ET=> );
			IF TON_C201.Q THEN
				Step_QuickScan:=210;
			END_IF
			
		210://7灯闪烁，机架运动到目标位置
			(*1.发送给上位机的数据*)
			WorkStation_TCP.PLC_SEND1.m_nMoveState:=0; //send [9]	//0-准备过程中 1-准备完成 2-曝光中 3-本次扫描结束
			TON_C201(IN:= FALSE);
			(*2.7灯闪烁*)
			GVL_State.bEnable_CTBOX:=TRUE;			//开启CTBOX发送灯使能
			LampCmd7:=E_LampCmd.慢闪;
			WorkStation_TCP.PLC_SEND1.m_nFocus:=7;	//按键提示0228
			
			(*3.旋转轴运动到目标位置*)
			Axis_XZ.XZ_AxisCmd.AxisPara.rAbsPosition:=LIMIT(-4,WorkStation_TCP.PLC_RECV1.m_nRotateBegin,363);
			Axis_XZ.XZ_AxisCmd.AxisPara.rAbsVelocity:=XZ_Velocity;
			
			IF WorkStation_TCP.PLC_RECV1.m_nSocketType=1 THEN
				Axis_XZ.XZ_AxisCmd.bAbs:=TRUE;
			END_IF;
			
			(*4.到位后2秒跳转*)
			TON_C210(IN:=ABS(Axis_XZ.XZ_AxisState.rActPosition-WorkStation_TCP.PLC_RECV1.m_nRotateBegin)<1 , PT:=T#1S , Q=> , ET=> );
			IF TON_C210.Q THEN
				Step_QuickScan:=221;	
			END_IF
		
		221://中间状态清零
			Axis_XZ.XZ_AxisCmd.bAbs:=FALSE;
			Axis_QJ.QJ_AxisCmd.bAbs:=FALSE;
			GVL_State.bEnable_CTBOX:=FALSE;//关闭CTBOX发送灯使能
			Step_QuickScan:=220;
			
		220://用户按7键，床自动走到预设位置
			(*1.按7键关闭7灯*)
			IF CTBOX_RS232.CTBOX_KEY_Manual THEN
				LampCmd7:=E_LampCmd.关闭;
				GVL_State.bEnable_CTBOX:=TRUE;//开启CTBOX发送灯使能
				WorkStation_TCP.PLC_SEND1.m_nFocus:=0;	//关闭按键提示0228
			END_IF
			
			(*2.触发床运动*)
			R_TRIG_C220(CLK:=CTBOX_RS232.CTBOX_KEY_Manual , Q=> );
			Axis_QJ.QJ_AxisCmd.AxisPara.rAbsPosition:=LIMIT(0,WorkStation_TCP.PLC_RECV1.m_fScanTop,900);
			Axis_QJ.QJ_AxisCmd.bAbs:=R_TRIG_C220.Q;
			
			(*3.跳转指令*)
			IF ABS(Axis_QJ.QJ_AxisState.rActPosition-WorkStation_TCP.PLC_RECV1.m_fScanTop)<1 AND (LampCmd7=E_LampCmd.关闭) THEN //保证必须按下7键
				WorkStation_TCP.PLC_SEND1.m_nMoveState:=1; //send [9]	//0-准备过程中 1-准备完成 2-曝光中 3-本次扫描结束
			ELSE
				WorkStation_TCP.PLC_SEND1.m_nMoveState:=0; //send [9]	//0-准备过程中 1-准备完成 2-曝光中 3-本次扫描结束
			END_IF
			
			(*4.延迟跳转，保证send [9]发送*)
			TOF_C80(IN:= FALSE);TON_C100(IN:=FALSE);TON_C90(IN:=FALSE);TON_C80(IN:=FALSE);TON_C70(IN:=FALSE);TON_C60(IN:=FALSE);
			TON_C210(IN:=FALSE);TON_C72(IN:=FALSE);TON_C201(IN:=FALSE);
			TON_C220(IN:=(WorkStation_TCP.PLC_SEND1.m_nMoveState=1) , PT:=T#2S , Q=> , ET=> );
			IF TON_C220.Q THEN
				Step_QuickScan:=70;
			END_IF		
	END_CASE
END_ACTION

ACTION _a_Debug_entry:


GVL_State.iPLC_State:=100;
END_ACTION

ACTION _a_Init_active:


InitMotor(); //电机初始化程序

GVL_State.iPLC_State:=10;

GVL_State.bEnable_CTBOX:=FALSE;
END_ACTION

ACTION _a_ScoutScan_active:


	CASE Step_Scout OF
		0:	//初始化准备流程
			(*1.给上位机发送的数据*)
			WorkStation_TCP.PLC_SEND1.m_nMoveState:=0;			//send[9]
			Axis_XZ.XZ_AxisCmd.bAbs:=FALSE;
			bTCP_Socket:=FALSE;
			bScoutLast := FALSE;
			
			(*2.运动准备数据*)
			(*2.1 写入旋转速度参数*)
			Axis_XZ.XZ_AxisCmd.AxisPara.rAbsVelocity:=36;//定位像扫描按照设定速度运动
			
			(*3.关闭CTBOX发送*)
			GVL_State.bEnable_CTBOX:=TRUE;//开启CTBOX发送灯的状态
			Step_Scout:=10;
		
		10:	//运动过程中变量复位标志
			TON_S30(IN:= FALSE );
			TON_S40(IN:= FALSE);TON_S50(IN:= FALSE);
			TON_S70(IN:= FALSE);TON_S80(IN:= FALSE);
			TOF_S50(IN:= FALSE);TON_S60(IN:= FALSE);
			TON_S52(IN:= FALSE );TON_S41(IN:=FALSE);
			TON_S43(IN:= FALSE );TON_S20_ABS(IN:=FALSE);
			Axis_XZ.XZ_AxisCmd.bAbs:=FALSE;
			Step_Scout:=20;
			
		20://开启运动
			(*1.给上位机发送的数据*)
			WorkStation_TCP.PLC_SEND1.m_nExpStates	:=1;//为曝光状态，枚举值，0:idle（空闲） 1:prep（训机） 2: ready（训机结束，准备完成，可以出束） 3: XrayOn（出射线） 4:XrayOff（关射线） 5 error；
			WorkStation_TCP.PLC_SEND1.m_nMoveState	:=0;//起始、终止状态， 默认值-1， 0为当前扫描方案（与常规意义不同，注意区别）处于准备好状态，可以准备扫描；1为当前扫描方案结束，运动过程中值为-1
			WorkStation_TCP.PLC_SEND1.m_nScanProType:=2;//执行扫描方案的类型，0为自动扫描，1为手动扫描，2为无设置意义的值，默认值为2
	
			(*2.旋转轴运动*)
			TON_S20_ABS(IN:= TRUE, PT:=T#1S );
			Axis_XZ.XZ_AxisCmd.bAbs:=TON_S20_ABS.Q;
			Axis_XZ.XZ_AxisCmd.AxisPara.rAbsPosition:=LIMIT(-4,WorkStation_TCP.PLC_RECV1.m_nRotateBegin,363);

			(*3.跳转下一个步骤*)	
			IF  ABS(Axis_XZ.XZ_AxisState.rActPosition-WorkStation_TCP.PLC_RECV1.m_nRotateBegin)<=1 THEN 
				Step_Scout:=21;
			END_IF
				
		21://射线源参数写入成功标志
			TON_S20_ABS(IN:=FALSE);
			Axis_XZ.XZ_AxisCmd.bAbs:=FALSE;
			IF XRAY_RS485.Standby_Step=60 THEN		(*增加射线源参数写入成功标志*)
				Step_Scout:=30;
			END_IF

		30: //开启7灯闪烁
			(*1.给上位机数据*)
			WorkStation_TCP.PLC_SEND1.m_nMoveState:=1;			//send[9]
			TON_S30(IN:=TRUE , PT:=T#1S , Q=> , ET=> );
			
			(*2.7灯闪烁*)
			GVL_State.bEnable_CTBOX:=TRUE;//开启CTBOX发送灯的状态
			LampCmd7:=E_LampCmd.慢闪;
			WorkStation_TCP.PLC_SEND1.m_nFocus:=7;//按键提示0228
			
			(*3.跳转*)
			IF TON_S30.Q THEN
				Step_Scout:=31;
			END_IF
			
		31:
			GVL_State.bEnable_CTBOX:=FALSE;//关闭CTBOX发送灯的状态
			Step_Scout:=40;
		
		40://等待用户按7键。此时7灯一直在闪烁
			(*1.发送上位机状态*)
			IF CTBOX_RS232.CTBOX_KEY_Manual THEN
				WorkStation_TCP.PLC_SEND1.m_nScanProType:=1;//执行扫描方案的类型，0为自动扫描，1为手动扫描，2为无设置意义的值，默认值为2
			END_IF
			
			(*2.7灯关闭*)
			TON_S41(IN:=(WorkStation_TCP.PLC_SEND1.m_nScanProType=1) , PT:=T#100MS , Q=> , ET=> );
			IF TON_S41.Q THEN
				LampCmd7:=E_LampCmd.关闭;  		//7灯关闭
				WorkStation_TCP.PLC_SEND1.m_nFocus:=0;//关闭按键提示0228
			END_IF
			
			TON_S42(IN:=FALSE , Q=> , ET=> );	//复位
			TON_S43(IN:=FALSE , Q=> , ET=> );	//复位
			
			(*3.跳转*)
			TON_S40(IN:= (WorkStation_TCP.PLC_SEND1.m_nScanProType=1), PT:=T#1S , Q=> , ET=> );
			IF TON_S40.Q THEN
				Step_Scout:=41;
			END_IF
			
		41://中间状态清零，特别是从80跳转过来的变量清零
			GVL_State.bEnable_CTBOX:=FALSE;//关闭CTBOX发送灯的状态
			TON_S41(IN:=FALSE);TON_S80(IN:=FALSE);
			Entity_IO.bXaryOne:=FALSE;
			GVL_SCAN.bEnableTrigger:=FALSE;
			GVL_State.bScoutSecond:=TRUE;
			IF XRAY_RS485.Standby_Step=60 THEN
				Step_Scout:=42;
			END_IF;	

		42:
			(*1.开启透视*)
			Entity_IO.bXaryOne:=TRUE;		//开启透视
			
			IF ABS(Axis_XZ.XZ_AxisState.rActPosition-WorkStation_TCP.PLC_RECV1.m_nAngleStart)<1 THEN
				GVL_SCAN.bEnableScout:=TRUE;	
			ELSE
				GVL_SCAN.bEnableScout:=FALSE;
			END_IF
			
			(*2.跳转指令*)
			TON_S43(IN:= Entity_IO.bXaryOne, PT:=T#1S , Q=> , ET=> );		//1秒
			IF TON_S43.Q THEN
				IF XRAY_RS485.Rad_Step>=20 THEN  //此时射线源收到  =20
					Step_Scout:=50;
				END_IF
			ELSE
			;
			END_IF;
			
			(*3.判断是否最后一次扫描标志位*)
			IF WorkStation_TCP.PLC_RECV1.m_nLastMsg=1 THEN
				bScoutLast := TRUE;
			ELSE
				bScoutLast := FALSE;
			END_IF 
			
			(*4.一二档信号超时报警，射线源30秒连续开启曝光会报警*)
			TON_S42(IN:=Entity_IO.bXaryOne , PT:=T#60S , Q=> , ET=> );
			IF TON_S42.Q THEN
				Step_Scout:=44;	
			END_IF
			
		44:
			Entity_IO.bXaryOne:=FALSE;
			GVL_SCAN.bJumpScan:=TRUE;		//结束扫描，射线源超时报警了，EL019，结束扫描
			Step_Scout:=44;	

		50://固定位置直接曝光4次
			TON_S43(IN:=FALSE , Q=> , ET=> );	//复位
			(*1.发送给上位机的数据*)
			WorkStation_TCP.PLC_SEND1.m_nMoveState	:=2;			//send[9]//0-准备过程中 1-准备完成 2-曝光中 3-本次扫描结束	
			WorkStation_TCP.PLC_SEND1.m_nScanProType:=2;			//send[16]
			
			(*2.开启允许曝光指令*)
			IF Entity_IO.bXaryOne AND ABS(Axis_XZ.XZ_AxisState.rActPosition-WorkStation_TCP.PLC_RECV1.m_nAngleStart)<1 THEN //新增射线源状态位置
				GVL_SCAN.bEnableTrigger:=TRUE;
			ELSE
				GVL_SCAN.bEnableTrigger:=FALSE;
			END_IF
			
			(*3.此过程给固定时间3秒,处理扫描*)
			TON_S50(IN:=TRUE , PT:=T#2S);
			IF TON_S50.Q THEN
				Step_Scout:=52;	
			END_IF
		
		52://出射线状态结束，采集射线源状态机信息 //增加2档信号8秒计时器清零操作
			TON_S52(IN:=NOT(Trigger_HaoboPannel.bScoutPulse) , PT:= T#3S );
			Entity_IO.bXaryOne:=NOT(TON_S52.Q);
			IF TON_S52.Q THEN
				IF XRAY_RS485.Main_Step=20 THEN
					Step_Scout:=60;
				END_IF
			END_IF
			
		60://判断是否最后一次扫描，如是，直接跳到待机模式，如果不是，接着定位扫描 ，第一次定位像和第二次定位像不一样，增加了床的运动
			TON_S80(IN:=FALSE);
			Entity_IO.bXaryOne:=FALSE;
			Axis_QJ.QJ_AxisCmd.bAbs:=FALSE;
			Axis_XZ.XZ_AxisCmd.bAbs:=FALSE;	
			TON_S70_ABSQ(IN:=FALSE);TON_S70_ABSX(IN:=FALSE);
			TON_S60(IN:=TRUE , PT:=T#1600MS , Q=> , ET=> );//留些时间给上位机发送本次扫描结束方案标志
			WorkStation_TCP.PLC_SEND1.m_nMoveState:=3;		//send[9] //0-准备过程中 1-准备完成 2-曝光中 3-本次扫描结束	
			IF TON_S60.Q THEN
				IF (WorkStation_TCP.PLC_RECV1.m_nCircleIndex+1)>=(WorkStation_TCP.PLC_RECV1.m_nCircleCount) AND bScoutLast THEN 	//用于区分自动扫是否最后一次，此时=1，=1都等于1
					GVL_SCAN.bJumpScan:=TRUE;
				END_IF;
			END_IF
			
			IF WorkStation_TCP.PLC_RECV1.m_nSocketType=1 THEN //增加第二次运动判断，m_nSocketType=1 
				Step_Scout:=70;
			END_IF
			
		70://上位机选择移动床位置，机架根据命令运动到位
			Axis_QJ.QJ_AxisCmd.AxisPara.rAbsPosition:=LIMIT(0,WorkStation_TCP.PLC_RECV1.m_fScanTop,900);
			Axis_QJ.QJ_AxisCmd.AxisPara.rAbsVelocity:=50; //单位mm/s
			TON_S70_ABSQ(IN:=TRUE , PT:=T#1S , Q=> , ET=> );
			Axis_QJ.QJ_AxisCmd.bAbs:=TON_S70_ABSQ.Q;
			
			Axis_XZ.XZ_AxisCmd.AxisPara.rAbsPosition:=LIMIT(-4,WorkStation_TCP.PLC_RECV1.m_nRotateBegin,363);
			TON_S70_ABSX(IN:=TRUE , PT:=T#1S , Q=> , ET=> );
			Axis_XZ.XZ_AxisCmd.bAbs:=TON_S70_ABSX.Q;
			
			IF ABS(Axis_QJ.QJ_AxisState.rActPosition-WorkStation_TCP.PLC_RECV1.m_fScanTop)<1 AND ABS(Axis_XZ.XZ_AxisState.rActPosition-WorkStation_TCP.PLC_RECV1.m_nRotateBegin)<1 THEN
				WorkStation_TCP.PLC_SEND1.m_nMoveState:=1;		//send[9] //0-准备过程中 1-准备完成 2-曝光中 3-本次扫描结束	
			ELSE
				WorkStation_TCP.PLC_SEND1.m_nMoveState:=0;		//send[9] //0-准备过程中 1-准备完成 2-曝光中 3-本次扫描结束	
			END_IF
			
			TON_S70(IN:=ABS(Axis_QJ.QJ_AxisState.rActPosition-WorkStation_TCP.PLC_RECV1.m_fScanTop)<1 
					AND ABS(Axis_XZ.XZ_AxisState.rActPosition-WorkStation_TCP.PLC_RECV1.m_nRotateBegin)<1, 
					PT:=T#2S , Q=> , ET=> );//给你2秒走到位
			IF TON_S70.Q THEN
				Step_Scout:=80;
			END_IF
		
		80://准备跳转，中间变量复位
			TOF_S50(IN:= FALSE);TON_S60(IN:= FALSE);TON_S70(IN:= FALSE);
			TON_S41(IN:= FALSE);TON_S42(IN:= FALSE);
			TON_S70_ABSQ(IN:=FALSE);TON_S70_ABSX(IN:=FALSE);
			Axis_QJ.QJ_AxisCmd.bAbs:=FALSE;
			Axis_XZ.XZ_AxisCmd.bAbs:=FALSE;
			TON_S80(IN:=TRUE , PT:= T#1S, Q=> , ET=> );
			IF TON_S80.Q THEN
				Step_Scout:=41;
			END_IF;	
	END_CASE
END_ACTION

ACTION _a_Logic_active:


//Entity_IO();
CTBOX_RS232();
WorkStation_TCP();
WorkMode();
XRAY_RS485();
//Trigger_HaoboPannel();

(*1.激光灯控制*)
(*按键后30秒自动停止输出，如果在30秒之内再次按键，下降沿有效，则立刻停止输出*)
	IF WorkMode.iWorkMode=99 THEN
		Entity_IO.bLaserOut:=bDebug_Laser;
	ELSE
		TP_Laser(IN:=Entity_IO.LeftPannel_LaserButton OR Entity_IO.RightPannel_LaserButton , PT:=T#5MS , Q=> , ET=> );
		R_TRIG1(CLK:=TP_Laser.Q , Q=> );
		TOF_Laser(IN:=TP_Laser.Q , PT:=T#60S , Q=> , ET=>TOF_ET );
		IF TOF_Laser.Q THEN
			IF R_TRIG1.Q THEN
				IF Entity_IO.bLaserOut THEN
					Entity_IO.bLaserOut:= FALSE;
				ELSE
					Entity_IO.bLaserOut:= TRUE;
				END_IF
			END_IF
		ELSE
			Entity_IO.bLaserOut:= FALSE;
		END_IF
	
		Entity_IO.bLeftPannel_LED2:=Entity_IO.bLaserOut;
		Entity_IO.bRightPannel_LED1:=Entity_IO.bLaserOut;
	END_IF

(*2.延迟断电功能*)
	TOF_PowerDelay(IN:= Entity_IO.bKeySwitch, PT:= T#5S, Q=> Entity_IO.bDelayPower);
	
(*3.TRIGGER*)
(*	iValidTrigger:=DINT_TO_UINT(Entity_IO.iEncoderPulse) MOD iHopeNumPulse;
	IF iValidTrigger>=0 AND iValidTrigger<=iHopeNumPulse/2  THEN
		Entity_IO.bTriggerOut:=TRUE;
	ELSE
		Entity_IO.bTriggerOut:=FALSE;	
	END_IF;
*)

(*4.中止扫描*)
	TON_StopScan(IN:= CTBOX_RS232.CTBOX_KEY_Stop, PT:= T#1S, Q=> , ET=> );
	
(*5.记录预设位置操作*)
	IF Entity_IO.LeftPannel_RecordPos OR Entity_IO.RightPannel_RecordPos THEN
		rBedRecordHeight:=Entity_IO.rRealPos;
		rBedRecordLength:=Axis_QJ.QJ_AxisState.rActPosition;
	ELSE
		rBedRecordHeight:=rBedRecordHeight;
		rBedRecordLength:=rBedRecordLength;
	END_IF
END_ACTION

ACTION _a_MoveXZ_active:
	
	CASE Step_XZ OF
		0:	//初始化准备流程
			(*1.给上位机发送的数据*)
			WorkStation_TCP.PLC_SEND1.m_nMoveState:=0;			//send[9]
			Axis_XZ.XZ_AxisCmd.bAbs:=FALSE;
			bTCP_Socket:=FALSE;
			bScoutLast := FALSE;
			
			(*2.运动准备数据*)
			(*2.1 写入旋转速度参数*)
			Axis_XZ.XZ_AxisCmd.AxisPara.rAbsVelocity:=18;//定位像扫描按照设定速度运动 改为18  0717
			
			Step_XZ:=10;
		
		10:	//运动过程中变量复位标志
			TON_S30(IN:= FALSE );
			TON_S20_ABS(IN:=FALSE);
			Axis_XZ.XZ_AxisCmd.bAbs:=FALSE;
			Step_XZ:=20;
			
		20://开启运动
			(*1.给上位机发送的数据*)
			WorkStation_TCP.PLC_SEND1.m_nExpStates	:=1;//为曝光状态，枚举值，0:idle（空闲） 1:prep（训机） 2: ready（训机结束，准备完成，可以出束） 3: XrayOn（出射线） 4:XrayOff（关射线） 5 error；
			WorkStation_TCP.PLC_SEND1.m_nMoveState	:=0;//起始、终止状态， 默认值-1， 0为当前扫描方案（与常规意义不同，注意区别）处于准备好状态，可以准备扫描；1为当前扫描方案结束，运动过程中值为-1
			WorkStation_TCP.PLC_SEND1.m_nScanProType:=2;//执行扫描方案的类型，0为自动扫描，1为手动扫描，2为无设置意义的值，默认值为2
	
			(*2.旋转轴运动*)
			TON_S20_ABS(IN:= TRUE, PT:=T#1S );
			Axis_XZ.XZ_AxisCmd.bAbs:=TON_S20_ABS.Q;
			Axis_XZ.XZ_AxisCmd.AxisPara.rAbsPosition:=180;		//固定走到0°改为180  0717

			(*3.跳转下一个步骤*)	
			IF  ABS(Axis_XZ.XZ_AxisState.rActPosition-WorkStation_TCP.PLC_RECV1.m_nRotateBegin)<=1 THEN 
				Step_XZ:=30;
			END_IF
			
		30:
			Axis_XZ.XZ_AxisCmd.bAbs:=FALSE;
			TON_S30(IN:= TRUE, PT:=T#1S );
			IF TON_S30.Q THEN
				Step_XZ:=40;
			END_IF
			
		40:
			GVL_SCAN.bJumpScan:=TRUE;		//跳出来了，哈哈
			
		END_CASE
END_ACTION

ACTION _a_SystemInfo_active:

	LS_GetIPAddress_1(
		xExecute:= bGetPLC_IP, 
		eNetPort:= 0, 
		xDone=> , 
		xError=> , 
		diErrorID=> , 
		byIpSegmengt1=> , 
		byIpSegmengt2=> , 
		byIpSegmengt3=> , 
		byIpSegmengt4=> );
	
	LS_SetIPAddress_1(
		xExecute:= bSetPLC_IP, 
		eNetPort:= 0, 
		byIpSegmengt1:= , 
		byIpSegmengt2:= , 
		byIpSegmengt3:= , 
		byIpSegmengt4:= , 
		xDone=> , 
		xError=> , 
		diErrorID=> );
	
	GetPLCLoad(xEnable:= TRUE, xValid=> , xError=> , diErrorID=> , fLoad=> rPLC_Load);
	
	LS_SetDintDT_1(
		xExecute:= bSetSysTime, 
		uiYear:= , 
		uiMonth:= , 
		uiDay:= , 
		uiHour:= , 
		uiMinute:= , 
		uiSecond:= , 
		xDone=> , 
		xError=> , 
		diErrorID=> );

	LS_ReadDintDT_1(
		xEnable:= TRUE, 
		xValid=> , 
		xError=> , 
		diErrorID=> , 
		uiYear=> , 
		uiMonth=> , 
		uiDay=> , 
		uiHour=> , 
		uiMinute=> , 
		uiSecond=> );
END_ACTION

ACTION _a_Debug_active:


(**)
IF WorkMode.iWorkMode=99 THEN
	Entity_IO.bXaryOne:=bTestXayOne;
	Entity_IO.bTriggerOut:=bTestTrigger;
	
	Entity_IO.bTriggerPannel:=bTestTrigger11;
	Entity_IO.bTriggerPannel_NOT:=bTestTrigger22;
ELSE
	;
END_IF


(*1.获取旋转编码器的数值*)
(*	EncoderNum1:=DINT_TO_UDINT(ABS(Entity_IO.iEncoderPulse));
	
	CASE iSamplingRate1 OF 
		360:
			iHopePulse1:=360;
		600:
			iHopePulse1:=216;//215
		1200:
			iHopePulse1:=108;
		2400:
			iHopePulse1:=54;//52
		ELSE
			iHopePulse1:=360;
	END_CASE
*)	
(*2.*)
(*	R_TRIG_debug(CLK:=WorkMode.iWorkMode=99 , Q=> );
	IF R_TRIG_debug.Q THEN
		iStartTrigger1:=EncoderNum1;
	END_IF
	
	DB_EncoderNum1:=ABS(EncoderNum1-iStartTrigger1);
	iValidTrigger:=UDINT_TO_UINT(DB_EncoderNum1) MOD iHopePulse1;
	
	IF (iValidTrigger)>=0 AND (iValidTrigger)<=iHopePulse1 / 2 THEN
			IF (iActNumPulse1)<=(iHopePulse1+2) THEN
				deubg_out:=TRUE;
				Entity_IO.bTriggerHaobo:=TRUE;
			ELSE
				deubg_out:=FALSE;
				Entity_IO.bTriggerHaobo:=FALSE;
			END_IF
	ELSE
		deubg_out:=FALSE;
		Entity_IO.bTriggerHaobo:=FALSE;
	END_IF
		
		(*-----------------------计数器清零操作-----------------------*)
	IF WorkMode.iWorkMode<>99 THEN
		iActNumPulse1:=0;
		deubg_out:=FALSE;
	END_IF

	R_TRIG_debug2(CLK:=(deubg_out), Q=> );
	IF R_TRIG1.Q THEN					(*计数一共输出多少脉冲*)
		iActNumPulse1:=iActNumPulse1+1;
	END_IF;
*)
END_ACTION

ACTION _a_ScoutDR_exit:



	LampCmd5:=E_LampCmd.关闭;
	LampCmd6:=E_LampCmd.关闭;
	LampCmd7:=E_LampCmd.关闭;
	LampCmd8:=E_LampCmd.关闭;
	
	GVL_SCAN.bEnableScout:=FALSE;
	
	Entity_IO.bTriggerPannel:=FALSE;
	Entity_IO.bTriggerOut:=FALSE;
END_ACTION

ACTION _a_Homing_exit:


	Axis_XZ.XZ_AxisCmd.bHome:=FALSE;
	Axis_QJ.QJ_AxisCmd.bHome:=FALSE;
END_ACTION

ACTION _a_ScoutDR_entry:



Step_DR:=0; 
GVL_State.iPLC_State:=55;
bTCP_Socket:=TRUE; //首次开机需要按2下开始采集
END_ACTION

TRANSITION T_Scout:


(*进入定位片扫描*)
	WorkStation_TCP.PLC_RECV1.m_nSocketType=1 AND WorkStation_TCP.PLC_RECV1.m_nExpId=1
END_TRANSITION

ACTION _a_Emergercy_active:


(*急停工作模式*)

(*1.所有电机下使能,升降电机禁止运动*)
	Axis_XZ.XZ_AxisCmd.bPower:=FALSE;//上使能
	Axis_QJ.QJ_AxisCmd.bPower:=FALSE;//上使能

	IF Entity_IO.bForceBrake THEN
		Entity_IO.bBrakeOut:=TRUE;//强制打开抱闸
	ELSE
		Entity_IO.bBrakeOut:=FALSE;//
	END_IF
	
	Motor_SJ(Enable:= FALSE);

(*2.射线源停止出束，一二档信号失能*)
	Entity_IO.bXaryTwo:=FALSE;
	Entity_IO.bXaryOne:=FALSE;
END_ACTION

END_PROGRAM

// Device/Application/Communication/CTBOX_RS232
PROGRAM CTBOX_RS232
VAR
	Open_0: COM.Open;
	Write_0: COM.Write;
	Read_0: COM.Read;
	Close_0: COM.Close;
	xOpen_Exe:BOOL;
	hComHandle:CAA.HANDLE;
	byWriteData:ARRAY [0..12] OF BYTE;
	xWrite_Exe:BOOL;
	xRead_Exe:BOOL;
    byReadData:ARRAY [0..15] OF BYTE;
    xClose_Exe:BOOL;
	aParamsB19200 : ARRAY [1..7] OF COM.PARAMETER := [
    (udiParameterId := COM.CAA_Parameter_Constants.udiPort,udiValue := 2), 					//指令端口2,3,4,5分别对应硬件接口com2、com0、com1、com3
    (udiParameterId := COM.CAA_Parameter_Constants.udiBaudrate,udiValue := 19200),			//波特率，设置为19200
    (udiParameterId := COM.CAA_Parameter_Constants.udiParity,udiValue := COM.PARITY.NONE),	//校验，设置为无校验
    (udiParameterId := COM.CAA_Parameter_Constants.udiStopBits,udiValue := COM.STOPBIT.ONESTOPBIT),//停止位，1位
    (udiParameterId := COM.CAA_Parameter_Constants.udiTimeout,udiValue := 500),				//超时时间，设置成500ms
    (udiParameterId := COM.CAA_Parameter_Constants.udiByteSize,udiValue := 8),				//数据位
    (udiParameterId := COM.CAA_Parameter_Constants.udiBinary, udiValue := 1)				//二进制参数，启用二进制模式
];		
	Check:UINT;//读取数据的和校验
	TON1,TON2:TON;//定时写入和读取数据
	TON3:Standard.TON;//延时打开串口
	TON_Reset:Standard.TON;
	i: INT;//
	CTBOX_KEY	:ARRAY [0..7] OF BOOL;
	Blink_Reset:Blink;
	Lamp5State,Lamp6State,Lamp7State,Lamp8State:BYTE;
	
	count: BYTE;
	bDebug_RS232:BOOL;
	A1,A2,A3,A4:BOOL;
	R_CLOSE:Standard.R_TRIG;
	bReset:BOOL;
	booting:BOOL:=TRUE;
	R_TRIG11:R_TRIG;
END_VAR

VAR_OUTPUT
	CTBOX_KEY_Manual		:BOOL;//手动扫描
	CTBOX_KEY_Auto			:BOOL;//自动扫描
	CTBOX_KEY_Stop			:BOOL;//中止扫描
	CTBOX_KEY_MoveDistance	:BOOL;//移动到扫描位置
	CTBOX_KEY_BedFore		:BOOL; //进床
	CTBOX_KEY_BedUp			:BOOL;//升床
	CTBOX_KEY_BedBack		:BOOL;//出床
	CTBOX_KEY_BedDown		:BOOL;//升床	
END_VAR

(*Readme*)
(*与CTbox进行通信*)
(*------------------------------------第一部分：RS232数据收发设置---------------------------------------*)
(*0.心跳*)
	IF R_TRIG11.Q THEN
		count:=count+1;
	END_IF;
	R_TRIG11(CLK:=Write_0.xDone , Q=> );
(*1.open*)
	IF booting AND TON3.Q  THEN
		bReset:=TRUE;
		booting:=FALSE;
	END_IF
	
	TON3(IN:=TRUE , PT:=T#10S);//开机后10秒打开串口
	Open_0(xExecute:=bReset , xDone=> , xBusy=> , xError=> , usiListLength:=20 , pParameterList:=ADR(aParamsB19200) , eError=> , hCom=>hComHandle );
	
(*2.Write*)
	TON1(IN:=NOT TON1.Q , PT:=T#58MS , Q=> , ET=> );
	Write_0(
			xExecute:= Open_0.xDone AND TON1.Q, //周期写入控制灯的命令，同时此命令也是查询CTBOX键值的命令，主动发才会回复键值
			xAbort:= , 
			udiTimeOut:=500 , 
			xDone=> , 
			xBusy=> , 
			xError=> , 
			xAborted=> , 
			hCom:= hComHandle, 
			pBuffer:= ADR(byWriteData), 
			szSize:= 12, 
			eError=> );	
	
		byWriteData[0]:=16#FD;
		byWriteData[1]:=16#F4;
		byWriteData[2]:=16#03;
		byWriteData[3]:=16#04;
		
		byWriteData[4]:=16+Lamp7State;
		byWriteData[5]:=32+Lamp8State;
		byWriteData[6]:=48+Lamp6State;
		byWriteData[7]:=64+Lamp5State;
		
		Check:=USINT_TO_UINT(byWriteData[0])+USINT_TO_UINT(byWriteData[1])+USINT_TO_UINT(byWriteData[2])+USINT_TO_UINT(byWriteData[3])+
					USINT_TO_UINT(byWriteData[4])+USINT_TO_UINT(byWriteData[5])+USINT_TO_UINT(byWriteData[6])+USINT_TO_UINT(byWriteData[7]);
		byWriteData[8]:=UINT_TO_USINT(Check MOD 256);   
		byWriteData[9]:=UINT_TO_USINT(Check / 256);
		byWriteData[10]:=16#4F;
		byWriteData[11]:=16#DF;
		
(*3.Read*)
	TON2(IN:=NOT TON2.Q , PT:=T#36MS , Q=> , ET=> );
	Read_0(
			xExecute:= Open_0.xDone AND TON2.Q AND NOT(xWrite_Exe), 
			xAbort:= , 
			udiTimeOut:= 500, 
			xDone=> , 
			xBusy=> , 
			xError=> , 
			xAborted=> , 
			hCom:= hComHandle, 
			pBuffer:= ADR(byReadData), 
			szBuffer:= 16, 
			eError=> , 
			szSize=> );
	
(*4.Close*)
	Close_0(
			xExecute:= xClose_Exe, 
			xDone=> , 
			xBusy=> , 
			xError=> , 
			hCom:= hComHandle, 
			eError=> );
			
(*5.Reset*)
(*	IF TON3.Q THEN			//开机10秒后在进行开始故障复位逻辑
		TON_Reset(IN:=(Read_0.szSize=0), PT:=T#2S , Q=> , ET=> ); 
		Blink_Reset(ENABLE:=TON_Reset.Q, TIMELOW:=T#5S , TIMEHIGH:=T#20MS , OUT=> );
		R_CLOSE(CLK:= TON_Reset.Q AND Blink_Reset.OUT, Q=> xClose_Exe);
		IF TON_Reset.Q AND Close_0.xDone THEN
			bReset:=TON_Reset.Q AND NOT(Blink_Reset.OUT);
		ELSE
			bReset:=TRUE;
		END_IF;
	END_IF			
*)		
(*---------------------------第二部分：数据处理---------------------------*)
(*2.1 数据接收处理*)
	IF byReadData[0]=16#FD AND byReadData[1]=16#F4 AND byReadData[2]=16#2 AND byReadData[3]=16#08 
		AND byReadData[14]=16#4F AND byReadData[15]=16#DF THEN	
		FOR i:=0 TO 7 BY 1 DO
			CTBOX_KEY[i]:=BYTE_TO_BOOL(byReadData[i+4]);
		END_FOR
	ELSE
		FOR i:=0 TO 7 BY 1 DO
    		CTBOX_KEY[i]:=FALSE;
		END_FOR
	END_IF
	

(*2.2.管脚分配*)
	CTBOX_KEY_Manual		:=CTBOX_KEY[0];		     
	CTBOX_KEY_Auto			:=CTBOX_KEY[1];			      
	CTBOX_KEY_Stop			:=CTBOX_KEY[2];			      
	CTBOX_KEY_MoveDistance	:=CTBOX_KEY[3];	
	CTBOX_KEY_BedFore		:=CTBOX_KEY[4];		    
	CTBOX_KEY_BedUp			:=CTBOX_KEY[5];			     
	CTBOX_KEY_BedBack		:=CTBOX_KEY[6];		    
	CTBOX_KEY_BedDown		:=CTBOX_KEY[7];	
	
(*3 数据发送处理*)
(*------5678四个灯状态处理-------------*)
	IF WorkMode.iWorkMode=99 AND bDebug_RS232 THEN		
		IF A1 THEN
			A2:=FALSE;
			A3:=FALSE;
			A4:=FALSE;
			Lamp5State:=16#00;
			Lamp6State:=16#00;
			Lamp7State:=16#00;
			Lamp8State:=16#00;
		ELSE
			IF A2 THEN
				A3:=FALSE;
				A4:=FALSE;
				Lamp5State:=16#02;
				Lamp6State:=16#02;
				Lamp7State:=16#02;
				Lamp8State:=16#02;
			ELSE
				IF A3 THEN
					A4:=FALSE;
					Lamp5State:=16#03;
					Lamp6State:=16#03;
					Lamp7State:=16#03;
					Lamp8State:=16#03;
				ELSE
					IF A4 THEN
						Lamp5State:=16#01;
						Lamp6State:=16#01;
						Lamp7State:=16#01;
						Lamp8State:=16#01;
					ELSE
						Lamp5State:=16#00;
						Lamp6State:=16#00;
						Lamp7State:=16#00;
						Lamp8State:=16#00;
					END_IF
				END_IF
			END_IF
		END_IF
	ELSE  //正常工作流程下的处理
		CASE PLC_PRG.LampCmd5 OF 
			E_LampCmd.关闭:Lamp5State:=16#00;
			E_LampCmd.常亮:Lamp5State:=16#01;
			E_LampCmd.慢闪:Lamp5State:=16#02;
			E_LampCmd.快闪:Lamp5State:=16#03;
			ELSE Lamp5State:=16#00;
		END_CASE
		
		CASE PLC_PRG.LampCmd6 OF 
			E_LampCmd.关闭:Lamp6State:=16#00;
			E_LampCmd.常亮:Lamp6State:=16#01;
			E_LampCmd.慢闪:Lamp6State:=16#02;
			E_LampCmd.快闪:Lamp6State:=16#03;
			ELSE Lamp6State:=16#00;
		END_CASE
		
			CASE PLC_PRG.LampCmd7 OF 
			E_LampCmd.关闭:Lamp7State:=16#00;
			E_LampCmd.常亮:Lamp7State:=16#01;
			E_LampCmd.慢闪:Lamp7State:=16#02;
			E_LampCmd.快闪:Lamp7State:=16#03;
			ELSE Lamp7State:=16#00;
		END_CASE
		
		CASE PLC_PRG.LampCmd8 OF 
			E_LampCmd.关闭:Lamp8State:=16#00;
			E_LampCmd.常亮:Lamp8State:=16#01;
			E_LampCmd.慢闪:Lamp8State:=16#02;
			E_LampCmd.快闪:Lamp8State:=16#03;
			ELSE Lamp8State:=16#00;
		END_CASE
	END_IF;

END_PROGRAM

// Device/Application/Logic/WorkMode
PROGRAM WorkMode

VAR
	count	:BYTE;	
	WorkModeTemp:INT:=22;//默认
	TON1,TON2	:TON;
	bDebugMode	:BOOL:=FALSE;
	booting:BOOL:=TRUE;


END_VAR

VAR_OUTPUT	
	iWorkMode	:INT;
END_VAR

(*Readme*)


	(*0.心跳*)
	count:=count+1;
	TON1(IN:= TRUE, PT:= T#10S, Q=> , ET=> );
	(*状态机切换逻辑，再复杂的话用if-condition方式*)
	IF (Entity_IO.bKeySwitch=FALSE) AND TON1.Q THEN			//记着取消NOT
		WorkModeTemp:=55;							//关机模式
		booting:=TRUE;
	ELSE
		IF bDebugMode THEN
			WorkModeTemp:=99;						//调试模式
		ELSE
			IF (Entity_IO.bEmergencyStop) THEN	//TRUE相当于被触发了
				WorkModeTemp:=33;					//急停模式
			ELSE
				IF Axis_XZ.XZ_AxisState.bAxisErr OR Axis_QJ.QJ_AxisState.bAxisErr THEN
					WorkModeTemp:=44;				//错误模式
				ELSE
					WorkModeTemp:=11;				//工作状态
				END_IF
			END_IF
		END_IF
	END_IF

	iWorkMode:=	WorkModeTemp;

END_PROGRAM

// Device/Application/Motor/Motor_SJ
PROGRAM Motor_SJ
VAR
	count		:BYTE;
//	bCalibrate	:BOOL;//标定
//	rZeroPos_TEMP: INT;
	TOF_Delay:TOF;//位置模式运动，超时后停止
	DB:REAL:=1.5;
END_VAR

VAR_INPUT
	Enable:BOOL;
END_VAR

VAR_OUTPUT	
//	rRealPos:REAL;
END_VAR

(*-----------------------------Readme---------------------------------*)
(*---------升降电机功能块---------------------------------------------*)
(*-------------输入管脚已有滤波---------------------------------------*)


(*0.心跳*)
	count:=count+1;
	
(*3.点动及位置控制，如果触碰到限位，首先手动移动到安全区域*)
	IF Enable THEN
		IF Entity_IO.bUpMotorMin THEN
			Entity_IO.bUpMotorNeg:=FALSE;
			IF (Entity_IO.LeftPannel_BedUp OR Entity_IO.RightPannel_BedUp OR CTBOX_RS232.CTBOX_KEY_BedUp)=TRUE AND (Entity_IO.LeftPannel_BedDown OR Entity_IO.RightPannel_BedDown OR CTBOX_RS232.CTBOX_KEY_BedDown)=FALSE THEN
				TOF_Delay(IN:=FALSE);//TOF复位
				Entity_IO.bUpMotorPos:=TRUE;
			END_IF;
		ELSE
			(*1.同时按了上升和下降*)
			IF (Entity_IO.LeftPannel_BedUp OR Entity_IO.RightPannel_BedUp OR CTBOX_RS232.CTBOX_KEY_BedUp) AND (Entity_IO.LeftPannel_BedDown OR Entity_IO.RightPannel_BedDown OR CTBOX_RS232.CTBOX_KEY_BedDown) THEN
				TOF_Delay(IN:=FALSE);//TOF复位
				Entity_IO.bUpMotorPos:=FALSE;
				Entity_IO.bUpMotorNeg:=FALSE;
			(*2.上升*)
			ELSIF (Entity_IO.LeftPannel_BedUp OR Entity_IO.RightPannel_BedUp OR CTBOX_RS232.CTBOX_KEY_BedUp)=TRUE 
					AND (Entity_IO.LeftPannel_BedDown=FALSE AND Entity_IO.RightPannel_BedDown=FALSE AND CTBOX_RS232.CTBOX_KEY_BedDown=FALSE) THEN
				TOF_Delay(IN:=FALSE);//TOF复位
				IF Entity_IO.rRealPos<=285 THEN
					Entity_IO.bUpMotorPos:=TRUE;
					Entity_IO.bUpMotorNeg:=FALSE;
				ELSE
					Entity_IO.bUpMotorPos:=FALSE;
					Entity_IO.bUpMotorNeg:=FALSE;
				END_IF
			(*3.下降*)
			ELSIF (Entity_IO.LeftPannel_BedUp=FALSE AND Entity_IO.RightPannel_BedUp=FALSE AND CTBOX_RS232.CTBOX_KEY_BedUp=FALSE) AND (Entity_IO.LeftPannel_BedDown OR Entity_IO.RightPannel_BedDown OR CTBOX_RS232.CTBOX_KEY_BedDown)=TRUE THEN
				TOF_Delay(IN:=FALSE);//TOF复位
				Entity_IO.bUpMotorPos:=FALSE;
				Entity_IO.bUpMotorNeg:=TRUE;
			(*4.上升下降都没按*)
			ELSE
				(*位置控制*)
				TOF_Delay(IN:=Entity_IO.LeftPannel_MoveRecordPos OR Entity_IO.RightPannel_MoveRecordPos , PT:=T#20S , Q=> , ET=> );//暂设20秒
				IF TOF_Delay.Q THEN //超时报警准备
					IF Entity_IO.rRealPos<(PLC_PRG.rBedRecordHeight-DB) THEN	
						Entity_IO.bUpMotorPos:=TRUE;
						Entity_IO.bUpMotorNeg:=FALSE;
					ELSIF Entity_IO.rRealPos>(PLC_PRG.rBedRecordHeight+DB) THEN	
						Entity_IO.bUpMotorPos:=FALSE;
						Entity_IO.bUpMotorNeg:=TRUE;
					ELSIF Entity_IO.rRealPos>=(PLC_PRG.rBedRecordHeight-DB) AND Entity_IO.rRealPos<=(PLC_PRG.rBedRecordHeight+DB) THEN
						Entity_IO.bUpMotorPos:=FALSE;
						Entity_IO.bUpMotorNeg:=FALSE;
					END_IF
				ELSE
					Entity_IO.bUpMotorPos:=FALSE;
					Entity_IO.bUpMotorNeg:=FALSE;
				END_IF
			END_IF
		END_IF
	ELSE
		Entity_IO.bUpMotorPos:=FALSE;
		Entity_IO.bUpMotorNeg:=FALSE;
	END_IF

END_PROGRAM

// Device/Application/Init/InitMotor
PROGRAM InitMotor
VAR
	sNameXZ,sNameQJ,sNameSJ: WSTRING:="";
END_VAR

(*Readme*)
(*电机初始化程序*)

(*1.电机名称*)
	sNameXZ:="旋转电机";
	sNameQJ:="前进电机";
	sNameSJ:="升降电机";
	
(*2.电机默认参数设置*)
	Axis_QJ.QJ_AxisCmd.AxisPara.rAbsVelocity:=60;
	Axis_QJ.QJ_AxisCmd.AxisPara.rAccDec:=25;
	Axis_QJ.QJ_AxisCmd.AxisPara.rJogVelocity:=60;
	Axis_QJ.QJ_AxisCmd.AxisPara.rRelVelocity:=30;
	
	Axis_XZ.XZ_AxisCmd.AxisPara.rAbsVelocity:=10;
	Axis_XZ.XZ_AxisCmd.AxisPara.rAccDec:=5;
	Axis_XZ.XZ_AxisCmd.AxisPara.rJogVelocity:=30;
	Axis_XZ.XZ_AxisCmd.AxisPara.rRelVelocity:=30;
	(*回零参数*)
	Axis_XZ.XZ_AxisCmd.AxisPara.rHomeHighSpeed:=30;
	Axis_XZ.XZ_AxisCmd.AxisPara.rHomeLowSpeed:=10;
	Axis_XZ.XZ_AxisCmd.AxisPara.rHomeAcc:=50;
	
	Axis_QJ.QJ_AxisCmd.AxisPara.rHomeHighSpeed:=30;
	Axis_QJ.QJ_AxisCmd.AxisPara.rHomeLowSpeed:=5;
	Axis_QJ.QJ_AxisCmd.AxisPara.rHomeAcc:=5;

END_PROGRAM

// Device/Application/BasicFBs/RC
FUNCTION_BLOCK RC
VAR_EXTERNAL

END_VAR

VAR_INPUT
	Input:UINT;
END_VAR
VAR_OUTPUT
	Output:UINT;
END_VAR
VAR
	prev:UINT;
END_VAR

(*======================== READ_ME ==============================*)
(*功能块：“低通滤波”                                           	 *)
(*=========================== END ===============================*)
prev:=UDINT_TO_UINT(6*UINT_TO_UDINT(Input)/10+4*UINT_TO_UDINT(prev)/10);
Output:=prev;

END_FUNCTION_BLOCK

// Device/Application/BasicFBs/Curve_Cs
FUNCTION_BLOCK Curve_Cs
VAR_EXTERNAL

END_VAR

VAR_INPUT
	X_Array	:ARRAY [ 0..9 ] OF INT;
	Y_Array	:ARRAY [ 0..9 ] OF INT;
	length	:INT;	
	Value_X	:INT;
END_VAR

VAR_OUTPUT
	Value_Y	:INT;
	Error:bool;
END_VAR

VAR
	BOOTING:BOOL:=0;
	POS_OR_NEG:bool;
	COUNT_NUM:INT:=0;
	COUNT_OLD:INT;
	TEMP_Length:INT;
END_VAR

(*============================ READ_ME ================================*)
(*功能块：“分段线性化曲线”                                           *)
(*根据给出的传感器分度表，进行分段线性计算，得出当前阻值对应的工程量   *)
(*注意，横坐标“X_Array”应从数组元素[0]开始按照从小到大的顺序写入值   *)
(*注意，length为写入数组元素的个数                                     *)
(*============================== END ==================================*)
	IF BOOTING=0 THEN
		IF ((X_Array[1]-X_Array[0])>0 AND (Y_Array[1]-Y_Array[0])>0) or ( (X_Array[1]-X_Array[0])<0 AND (Y_Array[1]-Y_Array[0])<0 ) THEN
			POS_OR_NEG:=1;
		ELSIF ((X_Array[1]-X_Array[0])>0 AND (Y_Array[1]-Y_Array[0])<0) or ( (X_Array[1]-X_Array[0])<0 AND (Y_Array[1]-Y_Array[0])>0 ) THEN
			POS_OR_NEG:=0;
		END_IF;		
		BOOTING:=1;
	END_IF;

	IF length<=1 or length>10 THEN
		TEMP_Length:=9;
	ELSE
		TEMP_Length:=length-1;
	END_IF;
	IF POS_OR_NEG=0 THEN
		IF COUNT_NUM<(TEMP_Length-1) THEN
			COUNT_NUM:=COUNT_NUM+1;
		ELSE
			COUNT_NUM:=0;
		END_IF;		
	ELSE
		IF COUNT_NUM>0 THEN
			COUNT_NUM:=COUNT_NUM-1;
		ELSE
			COUNT_NUM:=TEMP_Length-1;
		END_IF;		
	END_IF;
	COUNT_OLD:=COUNT_NUM+1;
	
	IF X_Array[COUNT_NUM]<X_Array[COUNT_OLD] and Error=0 THEN
		IF (Value_X>X_Array[COUNT_NUM]) AND (Value_X<=X_Array[COUNT_OLD]) THEN
			Value_Y:=Y_Array[COUNT_NUM]+dint_to_int(int_to_dint(Y_Array[COUNT_OLD]-Y_Array[COUNT_NUM])*int_to_dint(Value_X-X_Array[COUNT_NUM])/int_to_dint(X_Array[COUNT_OLD]-X_Array[COUNT_NUM]));
			IF POS_OR_NEG=1 THEN
				COUNT_NUM:=TEMP_Length-1;
			ELSE
				COUNT_NUM:=0;
			END_IF;				
		ELSIF Value_X<=X_Array[0] THEN
			Value_Y:=Y_Array[0];
		ELSIF Value_X>X_Array[TEMP_Length] THEN
			Value_Y:=Y_Array[TEMP_Length];		
		END_IF;	
	ELSE
		Error:=1;
		Value_Y:=0;
	END_IF;

END_FUNCTION_BLOCK

// Device/Application/BasicFBs/MeanValue
FUNCTION_BLOCK MeanValue
VAR_EXTERNAL

END_VAR

VAR_INPUT
	Input:UINT;
	PAR_Lenght:UINT;
	Reset:BOOL;
END_VAR
VAR_OUTPUT
	Output:UINT;
END_VAR
VAR
	Ka_Count:UINT:=1;
	Ka:UINT:=1;
	Ka_prev:UINT;
END_VAR

(*======================== READ_ME ==============================*)
(*功能块：“平均值滤波”                                         *)
(*=========================== END ===============================*)
	Ka:=UDINT_TO_UINT((UINT_TO_UDINT(Ka)*UINT_TO_UDINT(Ka_Count-1)+UINT_TO_UDINT(Input))/UINT_TO_UDINT(Ka_Count));
	Ka_Count:=Ka_count+1;
	IF(Reset OR Ka_count=PAR_Lenght+1) THEN
		Output:=Ka;
		Ka_Count:=1;
		Ka:=1;
	END_IF;

END_FUNCTION_BLOCK

// Device/Application/Refer/POU_CANopen
PROGRAM POU_CANopen
VAR
	
	MC_AxisConfi_CAN_0: MC_AxisConfi_CAN;
	ISV2_CAN6040_Axis_1:Str_LTCANopenAxis; //CANopen 轴结构体
	ControlWord AT%QW2 : UINT ;  //ControlWord地址
	StatusWord AT%IW2 : UINT ;  //StatusWord地址
	
	MC_Power_CAN_0: MC_Power_CAN;
	xPower: BOOL; //使能

	xAbsExecute: BOOL;  //启动绝对定位
	diPosition: DINT;   //目标位置
	udiVelocity: UDINT;  //目标速度
	udiAcceleration: UDINT; //目标加速度
	udiDeceleration: UDINT; //目标减速度
	
	
	xRelExecute: BOOL;//启动相对定位
	diDistance: DINT;   //相对距离
	
	
	MC_MoveVelocity_CAN_0: MC_MoveVelocity_CAN;
	xVelExecute: BOOL; //启动恒速运动
	Velocity: DINT;  //恒速运动目标速度
	Acceleration: UDINT;//恒速运动目标加速度
	Deceleration: UDINT;//恒速运动目标减速度
	
	MC_HomeSetPara_CAN_0: MC_HomeSetPara_CAN;
	MC_Home_CAN_0: MC_Home_CAN;
	xHomeSetPara: BOOL;  //设置回零参数
	xHome: BOOL;   //回零启动
	usiHomeMode: USINT;  //回零方式
	udiHomeHighSpeed: UDINT;  //回零高速度
	udiHomeLowSpeed: UDINT;    //回零低速度
	udiHomeAcceleration: UDINT;   //回零加速度
	
	MC_Stop_CAN_0: MC_Stop_CAN;
	xStop: BOOL;  //紧急停止
	
	MC_Reset_CAN_0: MC_Reset_CAN;
	xReset: BOOL; //清除错误
	
	MC_WriteODPara_CAN_0: MC_WriteODPara_CAN;
	MC_ReadODPara_CAN_0: MC_ReadODPara_CAN;
	xWriteODPara: BOOL; //写对象字典参数
	xReadODPara: BOOL; //读对象字典参数
	Index: WORD;  //索引
	SubIndex: BYTE;  //子索引
	Data: ARRAY [0..3] OF BYTE;  //写入数据
	DataLength: USINT;  //写入数据长度
	
	MC_JOG_CAN_0: MC_JOG_CAN;
	JogForward: BOOL ;  //正向点动
	JogBackword: BOOL;  //反向点动
	MC_MoveAbsoluteIme_CAN_0: MC_MoveAbsoluteIme_CAN;
	MC_MoveRelativeIme_CAN_0: MC_MoveRelativeIme_CAN;
	MC_Halt_CAN_0: MC_Halt_CAN;
	MC_ReadStatus_CAN_0: MC_ReadStatus_CAN;
	
	AA: POINTER TO _3SCOS.CANRemoteDevice_Diag;   //从站ISV2_CAN6040的地址
	B: _3SCOS.DEVICE_STATE;    //从站ISV2_CAN6040状态
	C: BYTE;  //从站ISV2_CAN6040的节点ID
	posi: UDINT;
END_VAR



A01_MC_AxisConfi();  		//根据节点ID 将CANopen轴 与 CANopen对应从站 进行绑定
A02_MC_Power();  			//CANopen轴使能
A03_MC_MoveAbsolute();   	//CANopen轴绝对定位
A04_MC_MoveRelative();   	//CANopen轴相对定位
A05_MC_MoveVelocity();   	//CANopen轴恒速运动
A06_MC_Home();   			//CANopen轴回零
A07_MC_Stop();   			//CANopen轴紧急停止
A08_MC_Reset();  	 		//CANopen轴清除错误
A09_ODPara();   			//CANopen轴读写对象字典参数
A10_MC_JOG();    			//CANopen轴JOG点动运动
A11_MC_ReadStatus_CAN();     //CANopen轴读轴状态

// 可通过 ISV2_CAN6040.CANopenState 状态监测从站 ISV2_CAN6040 是否掉线

AA :=ADR(CANopen_Device_XZ);
B := AA^.CANopenState;
C := AA^.NodeID ;

ACTION A01_MC_AxisConfi:
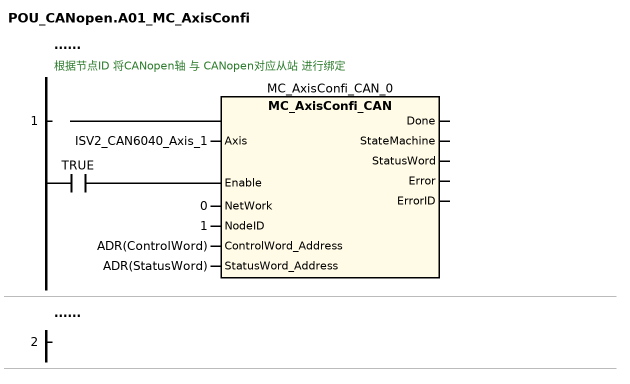
// NETWORK 1: ......
// 根据节点ID 将CANopen轴 与 CANopen对应从站 进行绑定
MC_AxisConfi_CAN_0(
    Axis := ISV2_CAN6040_Axis_1,
    Enable := TRUE,
    NetWork := 0,
    NodeID := 1,
    ControlWord_Address := ADR(ControlWord),
    StatusWord_Address := ADR(StatusWord)); // MC_AxisConfi_CAN

// NETWORK 2: ......
END_ACTION

ACTION A04_MC_MoveRelative:
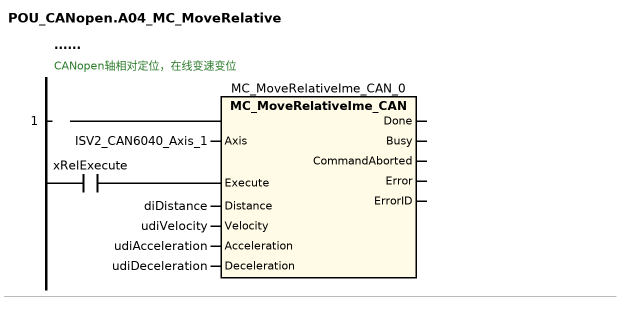
// NETWORK 1: ......
// CANopen轴相对定位，在线变速变位
MC_MoveRelativeIme_CAN_0(
    Axis := ISV2_CAN6040_Axis_1,
    Execute := xRelExecute,
    Distance := diDistance,
    Velocity := udiVelocity,
    Acceleration := udiAcceleration,
    Deceleration := udiDeceleration); // MC_MoveRelativeIme_CAN
END_ACTION

ACTION A02_MC_Power:
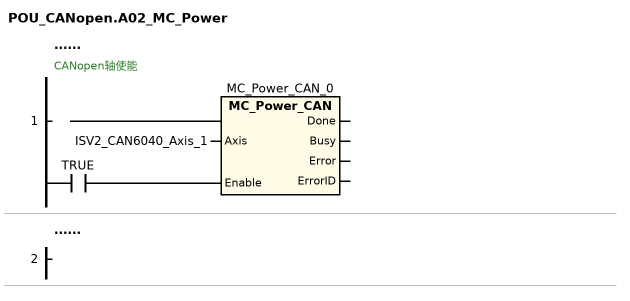
// NETWORK 1: ......
// CANopen轴使能
MC_Power_CAN_0(Axis := ISV2_CAN6040_Axis_1, Enable := TRUE); // MC_Power_CAN

// NETWORK 2: ......
END_ACTION

ACTION A09_ODPara:
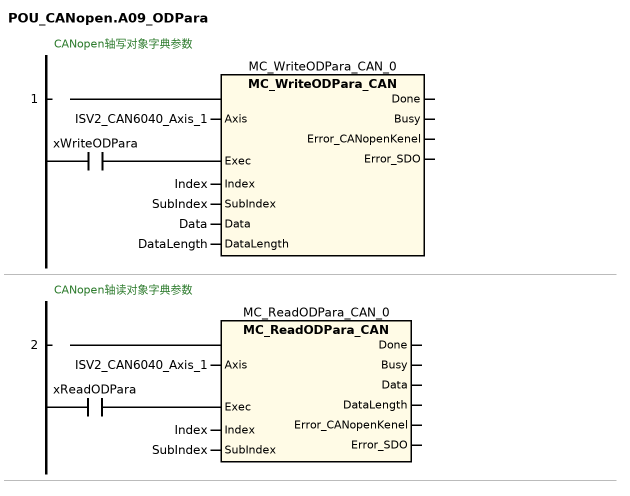
// NETWORK 1
// CANopen轴写对象字典参数
MC_WriteODPara_CAN_0(
    Axis := ISV2_CAN6040_Axis_1,
    Exec := xWriteODPara,
    Index := Index,
    SubIndex := SubIndex,
    Data := Data,
    DataLength := DataLength); // MC_WriteODPara_CAN

// NETWORK 2
// CANopen轴读对象字典参数
MC_ReadODPara_CAN_0(Axis := ISV2_CAN6040_Axis_1, Exec := xReadODPara, Index := Index, SubIndex := SubIndex); // MC_ReadODPara_CAN
END_ACTION

ACTION A03_MC_MoveAbsolute:
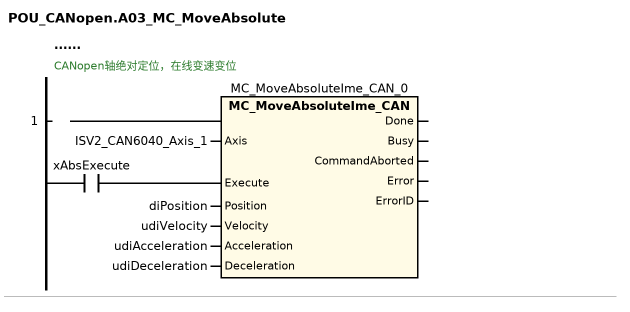
// NETWORK 1: ......
// CANopen轴绝对定位，在线变速变位
MC_MoveAbsoluteIme_CAN_0(
    Axis := ISV2_CAN6040_Axis_1,
    Execute := xAbsExecute,
    Position := diPosition,
    Velocity := udiVelocity,
    Acceleration := udiAcceleration,
    Deceleration := udiDeceleration); // MC_MoveAbsoluteIme_CAN
END_ACTION

ACTION A06_MC_Home:
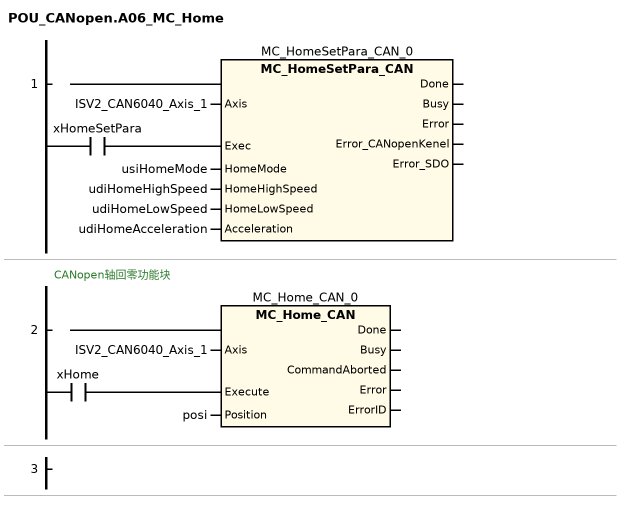
// NETWORK 1
MC_HomeSetPara_CAN_0(
    Axis := ISV2_CAN6040_Axis_1,
    Exec := xHomeSetPara,
    HomeMode := usiHomeMode,
    HomeHighSpeed := udiHomeHighSpeed,
    HomeLowSpeed := udiHomeLowSpeed,
    Acceleration := udiHomeAcceleration); // MC_HomeSetPara_CAN

// NETWORK 2
// CANopen轴回零功能块
MC_Home_CAN_0(Axis := ISV2_CAN6040_Axis_1, Execute := xHome, Position := posi); // MC_Home_CAN

// NETWORK 3
END_ACTION

ACTION A10_MC_JOG:
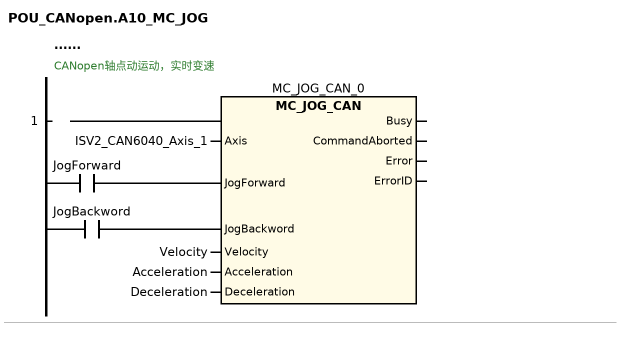
// NETWORK 1: ......
// CANopen轴点动运动，实时变速
MC_JOG_CAN_0(
    Axis := ISV2_CAN6040_Axis_1,
    JogForward := JogForward,
    JogBackword := JogBackword,
    Velocity := Velocity,
    Acceleration := Acceleration,
    Deceleration := Deceleration); // MC_JOG_CAN
END_ACTION

ACTION A11_MC_ReadStatus_CAN:
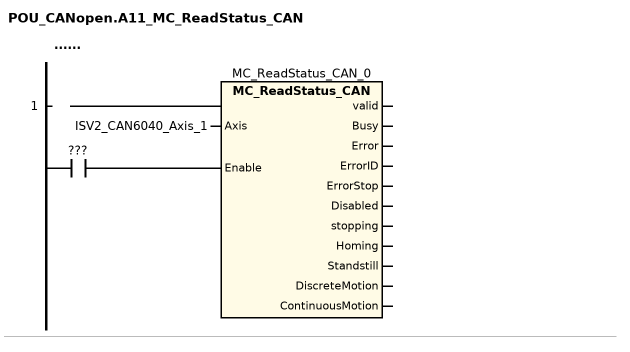
// NETWORK 1: ......
MC_ReadStatus_CAN_0(Axis := ISV2_CAN6040_Axis_1); // MC_ReadStatus_CAN
END_ACTION

ACTION A08_MC_Reset:
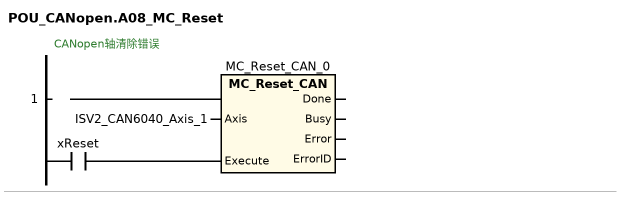
// NETWORK 1
// CANopen轴清除错误
MC_Reset_CAN_0(Axis := ISV2_CAN6040_Axis_1, Execute := xReset); // MC_Reset_CAN
END_ACTION

ACTION A07_MC_Stop:
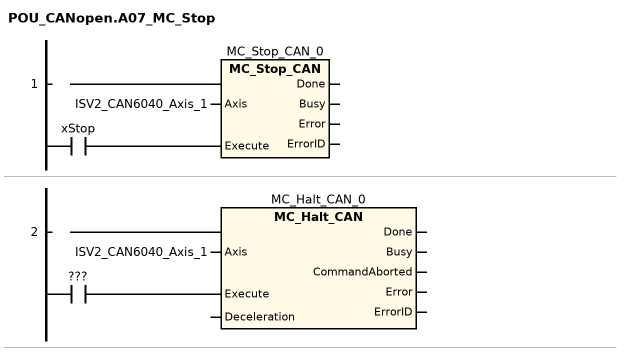
// NETWORK 1
MC_Stop_CAN_0(Axis := ISV2_CAN6040_Axis_1, Execute := xStop); // MC_Stop_CAN

// NETWORK 2
MC_Halt_CAN_0(Axis := ISV2_CAN6040_Axis_1); // MC_Halt_CAN
END_ACTION

ACTION A05_MC_MoveVelocity:
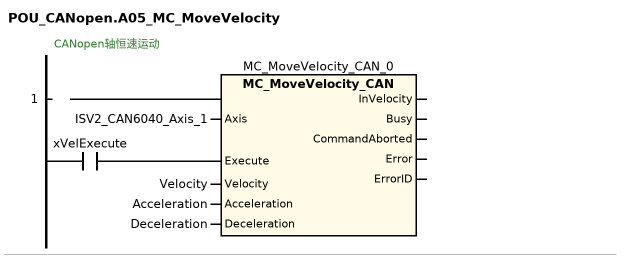
// NETWORK 1
// CANopen轴恒速运动
MC_MoveVelocity_CAN_0(
    Axis := ISV2_CAN6040_Axis_1,
    Execute := xVelExecute,
    Velocity := Velocity,
    Acceleration := Acceleration,
    Deceleration := Deceleration); // MC_MoveVelocity_CAN
END_ACTION

END_PROGRAM

// Device/Application/BasicFBs/Cut
FUNCTION_BLOCK Cut     (*把输入值进行预处理，调整斜率，消除两端的非线性影响*)
VAR_INPUT
	Input:UINT;
	PAR_InputlLowLimit:UINT;               (*此值的取值范围为0-255，一般在0—50之间*)
	PAR_InputHighLimit:UINT;               (*此值的取值范围为0-255，一般在200-255之间*)
END_VAR
VAR_OUTPUT
	Output:UINT;
	LowLimit:BOOL;
	HighLimit:BOOL;
END_VAR
VAR
END_VAR

(*功能描述：
把输入值进行预处理，调整斜率，消除两端非线性影响。
输入参数：
（1）Input，UINT型，要处理的信号。
（2）PAR_InputILowLimit，UINT型，用来控制输出的下限。当Input<=256*PAR_InputILowLimit时输出为0。
（3）PAR_InputHighLimit，UINT型，用来控制输出的上限。当Input>=256*PAR_InputHighLimit时输出就为256*PAR_InputHighLimit。
输出参数：
（1）Output，UINT型，处理完的信号。
（2）LowLimit，BOOL型，Input<=256*PAR_InputILowLimit时LowLimit为TRUE。
（3）HighLimit，BOOL型，Input>=256*PAR_InputHighLimit时HighLimit为TRUE。
*)

	LowLimit:=0;
	HighLimit:=0;
	PAR_InputlLowLimit:=PAR_InputlLowLimit*256;
	PAR_InputHighLimit:=PAR_InputHighLimit*256;
	IF(Input>=PAR_InputHighLimit) THEN
		Output:=0;
		HighLimit:=1;
	ELSIF(Input<=PAR_InputlLowLimit) THEN
		Output:=0;
		LowLimit:=1;
	ELSE
		Output:=DWORD_TO_UINT((Input-PAR_InputlLowLimit)*65536/(65536-PAR_InputlLowLimit-(65535-PAR_InputHighLimit)));
	END_IF

END_FUNCTION_BLOCK

// Device/Application/Logic/Trigger_YrayPannel
PROGRAM Trigger_YrayPannel
VAR
	count:BYTE;
	booting:BOOL:=TRUE;
	iHopePulse:UINT;
	EncoderNum:UDINT;
	iValidTrigger:UINT;
	NumTrigger:BYTE:=4;
	
	TOF_Trig,TOF_Scout:Standard.TOF;
	Blink_Scout:Blink;
	F_TRIG1:Standard.F_TRIG;
	R_TRIG1:Standard.R_TRIG;
END_VAR

VAR_INPUT
	iSamplingRate:UINT;
	bEnableTrigger:BOOL;
	bEnableScout:BOOL;
END_VAR

VAR_OUTPUT	
	iActNumPulse:UINT;//有效触发次数
	bScoutPulse:BOOL;
END_VAR

(*README*)
(*脉冲触发信号处理*)

(*0.心跳*)
	count:=count+1;
	
(*1.初始化函数*)
	IF booting THEN
		booting:=FALSE;
	END_IF
	
(*2.获取上位机发送的采样率*)//
	iSamplingRate:=UDINT_TO_UINT(WorkStation_TCP.PLC_RECV1.m_nSamplingRate);//采样率，有4个选项：2400帧/圈；1200帧/圈；600帧/圈,360帧/圈 recv[21]
	
(*3.处理多少个脉冲输出一个trigger*)
	CASE iSamplingRate OF 
		360:
			iHopePulse:=360;
		600:
			iHopePulse:=215;
		1200:
			iHopePulse:=108;
		2400:
			iHopePulse:=52;
		ELSE
			iHopePulse:=360;
	END_CASE
	
(*4.获取旋转编码器的数值*)
	EncoderNum:=DINT_TO_UDINT(ABS(Entity_IO.iEncoderPulse));
	
(*5.有效的输出的脉冲，50%的占空比*)
	iValidTrigger:=UDINT_TO_UINT(EncoderNum) MOD iHopePulse;
	
(*6.主逻辑，分2个工作模式，1是根据CBCT角度旋转触发，一个是根据定位像连续触发三次，次数可设*)
	TOF_Trig(IN:= GVL_SCAN.bEnableTrigger, PT:=T#1S , Q=> , ET=> 	);	//使能触发
	TOF_Scout(IN:= GVL_SCAN.bEnableScout,  PT:=T#1S , Q=> , ET=> 	);	//定位像自动触发标志
	IF TOF_Trig.Q AND Entity_IO.bXaryOne THEN
		(*--------------------------CBCT扫描，根据角度输出曝光指令-------------------------------*)
		IF GVL_State.iPLC_State=60 THEN  
			IF (iValidTrigger)>=0 AND (iValidTrigger)<=iHopePulse / 2 THEN
				IF (iActNumPulse)<=(iSamplingRate+2) THEN
					Entity_IO.bTriggerOut:=TRUE;
					Entity_IO.bTriggerPannel_NOT:=TRUE;
				ELSE
					Entity_IO.bTriggerOut:=FALSE;
					Entity_IO.bTriggerPannel_NOT:=FALSE;
				END_IF
			ELSE
				Entity_IO.bTriggerOut:=FALSE;
				Entity_IO.bTriggerPannel_NOT:=FALSE;
			END_IF
			
			(*-----------------------计数器清零操作-----------------------*)
			IF PLC_PRG.Step_CBCT<=70 THEN
				iActNumPulse:=0;
				Entity_IO.bTriggerOut:=FALSE;
				Entity_IO.bTriggerPannel_NOT:=FALSE;
			END_IF
		END_IF	
		(*-------------------------定位像扫描，固定角度直接曝光4次--------------------------------*)
		IF GVL_State.iPLC_State=50 THEN
			IF TOF_Scout.Q=TRUE THEN
			(*-----------------三个以内正常输出------曝光4次----------------------*)
				IF iActNumPulse<NumTrigger THEN
					Blink_Scout(ENABLE:= TRUE, TIMELOW:=T#200MS , TIMEHIGH:=T#10MS , OUT=> );//TIMEHIGH 的时间要小于曝光时间，当前曝光时间是20ms
					Entity_IO.bTriggerOut:=Blink_Scout.OUT;
					Entity_IO.bTriggerPannel_NOT:=Blink_Scout.OUT;
					bScoutPulse:=TRUE;			//定位像曝光中
				ELSE
					Blink_Scout(ENABLE:= FALSE);
					Entity_IO.bTriggerOut:=FALSE;
					Entity_IO.bTriggerPannel_NOT:=FALSE;
					bScoutPulse:=FALSE;
				END_IF
			ELSE
				Blink_Scout(ENABLE:= FALSE);
				Entity_IO.bTriggerOut:=FALSE;
				Entity_IO.bTriggerPannel_NOT:=FALSE;
				bScoutPulse:=FALSE;
			END_IF
		END_IF
		
	ELSE
		Entity_IO.bTriggerOut:=FALSE;
		Entity_IO.bTriggerPannel_NOT:=FALSE;
	END_IF
	
	(*-----------------计数一共有多少个脉冲输出--------------------*)
	R_TRIG1(CLK:=(Entity_IO.bTriggerOut) AND (GVL_State.iPLC_State=50 OR GVL_State.iPLC_State=60) AND (PLC_PRG.Step_Scout<>42)  , Q=> );
	IF R_TRIG1.Q THEN					(*计数一共输出多少脉冲*)
		iActNumPulse:=iActNumPulse+1;
	END_IF;

(*7.探测器反向输出*)
	Entity_IO.bTriggerPannel:=NOT(Entity_IO.bTriggerPannel_NOT);
	
